KUKA KRL program: EPS_2_251825_SA13_A_20260116064054.src

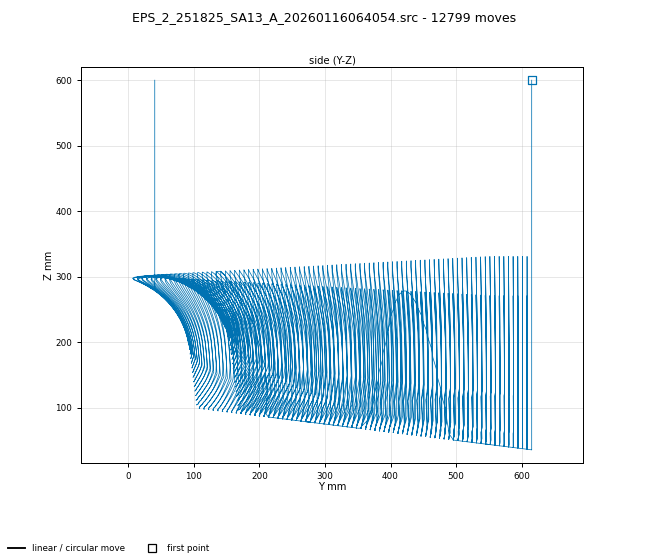
[picture p0: tool path of EPS_2_251825_SA13_A_20260116064054.src, 12799 of 12801 moves have a stored position in this frame; points joined in program order, loops and branches not executed]
&ACCESS RVP
&REL 4
&COMMENT QRS 19112012
&PARAM EDITMASK = *
DEF PART()
EXT BAS (BAS_COMMAND :IN,REAL :IN )
INT I
BAS (#INITMOV,0 )

;KUKA QRS Post kuka4.cps  Date:22-06-2017 !

File_ID=2975

QRS_PRE_INIT()

;Init var - Until changes are made in qrs_pre_init
Outlet_Square_prg=0
Inlet_1_Square_prg=0
Inlet_2_Square_prg=0
Inlet_3_Square_prg=0
Inlet_4_Square_prg=0
Inlet_5_Square_prg=0

Outlet_1={X 0.000, Y 551.740, Z 230.500, B 0.000, E1 0.000 }
Inlet_1={X 0.000, Y 556.010, Z 170.500, B 0.000, E1 170.000 }
Outlet_1_type=201
Inlet_1_type=201
;QRS#1=Sidecore dimensions
;QRS#2=200-8" PVC SDR 35
;QRS#3=200-8" PVC SDR 35
;QRS#4=
;QRS#5=
;QRS#6=
;QRS#7=
;QRS#8=
;QRS#9=12-08 PSX
;QRS#10=12-08 PSX
;QRS#11=
;QRS#12=
;QRS#13=
;QRS#14=
;QRS#15=
;QRS#16=1220x127x610 2'
;QRS#17=EPS Height
;QRS#18=331
;QRS#19=*
;QRS#20= UPDATED VERSION 22-06-2017
;QRS#21=*
Outlet_Square=0100
Inlet_1_Square=0100
Inlet_2_Square=0
Inlet_3_Square=0
Inlet_4_Square=0
Inlet_5_Square=0
Mill_Square=1
Outlet_Square_Prg=204
Inlet_1_Square_prg=204

QRS_INIT()

$ADVANCE=5

; T1
PTP {E1 173.62,E2 173.62}
PTP {X 0,Y 615.489,A -85,B 0,C 180,E1 173.62,E2 173.62,E3 0,E4 0,E5 0,E6 0}
QRS_SPEED_INIT()
LIN {X 0,Y 615.489,Z 600,A -85,B 0,C 180,E1 173.62,E2 173.62,E3 0,E4 0,E5 0,E6 0} C_VEL
LIN {X 0,Y 615.489,Z 45.866,A -85,B 0,C 180,E1 173.62,E2 173.62} C_VEL
LIN {X 0,Y 615.489,Z 37.686,A -85,B 0,C 180,E1 173.62,E2 173.62} C_VEL
LIN {X 0,Y 615.477,Z 35.686,A -85,B 0,C 180,E1 173.434,E2 173.434} C_VEL
LIN {X 0,Y 615.485,Z 35.695,A -85,B 0,C 180,E1 170.801,E2 170.801} C_VEL
LIN {X 0,Y 615.464,Z 35.693,A -85,B 0,C 180,E1 168.139,E2 168.139} C_VEL
LIN {X 0,Y 615.491,Z 35.685,A -85,B 0,C 180,E1 165.451,E2 165.451} C_VEL
LIN {X 0,Y 615.483,Z 35.698,A -85,B 0,C 180,E1 162.729,E2 162.729} C_VEL
LIN {X 0,Y 615.474,Z 35.687,A -85,B 0,C 180,E1 159.967,E2 159.967} C_VEL
LIN {X 0,Y 615.488,Z 35.701,A -85,B 0,C 180,E1 157.156,E2 157.156} C_VEL
LIN {X 0,Y 615.46,Z 35.69,A -85,B 0,C 180,E1 154.437,E2 154.437} C_VEL
LIN {X 0,Y 615.491,Z 35.695,A -85,B 0,C 180,E1 151.55,E2 151.55} C_VEL
LIN {X 0,Y 615.46,Z 35.694,A -85,B 0,C 180,E1 148.919,E2 148.919} C_VEL
LIN {X 0,Y 615.467,Z 35.688,A -85,B 0,C 180,E1 146.469,E2 146.469} C_VEL
LIN {X 0,Y 615.483,Z 35.701,A -85,B 0,C 180,E1 143.575,E2 143.575} C_VEL
LIN {X 0,Y 615.454,Z 35.692,A -85,B 0,C 180,E1 140.942,E2 140.942} C_VEL
LIN {X 0,Y 615.481,Z 35.687,A -85,B 0,C 180,E1 138.526,E2 138.526} C_VEL
LIN {X 0,Y 615.485,Z 35.699,A -85,B 0,C 180,E1 135.85,E2 135.85} C_VEL
LIN {X 0,Y 615.45,Z 35.692,A -85,B 0,C 180,E1 133.248,E2 133.248} C_VEL
LIN {X 0,Y 615.488,Z 35.69,A -85,B 0,C 180,E1 130.607,E2 130.607} C_VEL
LIN {X 0,Y 615.468,Z 35.698,A -85,B 0,C 180,E1 128.01,E2 128.01} C_VEL
LIN {X 0,Y 615.446,Z 35.694,A -85,B 0,C 180,E1 125.619,E2 125.619} C_VEL
LIN {X 0,Y 615.463,Z 35.69,A -85,B 0,C 180,E1 123.238,E2 123.238} C_VEL
LIN {X 0,Y 615.49,Z 35.692,A -85,B 0,C 180,E1 120.92,E2 120.92} C_VEL
LIN {X 0,Y 615.47,Z 35.699,A -85,B 0,C 180,E1 118.447,E2 118.447} C_VEL
LIN {X 0,Y 615.47,Z 35.794,A -85,B 0,C 180,E1 117.293,E2 117.293} C_VEL
LIN {X 0,Y 615.455,Z 50.485,A -85,B 0,C 180,E1 114.633,E2 114.633} C_VEL
LIN {X 0,Y 615.477,Z 60.616,A -85,B 0,C 180,E1 112.814,E2 112.814} C_VEL
LIN {X 0,Y 615.485,Z 166.964,A -85,B 0,C 180,E1 111.542,E2 111.542} C_VEL
LIN {X 0,Y 615.489,Z 179.954,A -85,B 0,C 180,E1 111.256,E2 111.256} C_VEL
LIN {X 0,Y 615.494,Z 193.256,A -85,B 0,C 180,E1 110.818,E2 110.818} C_VEL
LIN {X 0,Y 615.466,Z 204.889,A -85,B 0,C 180,E1 110.294,E2 110.294} C_VEL
LIN {X 0,Y 615.47,Z 215.474,A -85,B 0,C 180,E1 109.686,E2 109.686} C_VEL
LIN {X 0,Y 615.499,Z 226.345,A -85,B 0,C 180,E1 108.905,E2 108.905} C_VEL
LIN {X 0,Y 615.496,Z 235.253,A -85,B 0,C 180,E1 108.119,E2 108.119} C_VEL
LIN {X 0,Y 615.496,Z 244.551,A -85,B 0,C 180,E1 107.099,E2 107.099} C_VEL
LIN {X 0,Y 615.496,Z 251.406,A -85,B 0,C 180,E1 106.169,E2 106.169} C_VEL
LIN {X 0,Y 615.497,Z 257.042,A -85,B 0,C 180,E1 105.226,E2 105.226} C_VEL
LIN {X 0,Y 615.496,Z 261.719,A -85,B 0,C 180,E1 104.242,E2 104.242} C_VEL
LIN {X 0,Y 615.497,Z 265.484,A -85,B 0,C 180,E1 103.201,E2 103.201} C_VEL
LIN {X 0,Y 615.494,Z 267.337,A -85,B 0,C 180,E1 102.53,E2 102.53} C_VEL
LIN {X 0,Y 615.496,Z 268.704,A -85,B 0,C 180,E1 101.861,E2 101.861} C_VEL
LIN {X 0,Y 615.496,Z 270.232,A -85,B 0,C 180,E1 100.527,E2 100.527} C_VEL
LIN {X 0,Y 615.498,Z 270.372,A -85,B 0,C 180,E1 99.862,E2 99.862} C_VEL
LIN {X 0,Y 615.496,Z 269.451,A -85,B 0,C 180,E1 98.537,E2 98.537} C_VEL
LIN {X 0,Y 615.495,Z 268.407,A -85,B 0,C 180,E1 97.876,E2 97.876} C_VEL
LIN {X 0,Y 615.495,Z 265.082,A -85,B 0,C 180,E1 96.583,E2 96.583} C_VEL
LIN {X 0,Y 615.496,Z 261.297,A -85,B 0,C 180,E1 95.57,E2 95.57} C_VEL
LIN {X 0,Y 615.498,Z 256.495,A -85,B 0,C 180,E1 94.584,E2 94.584} C_VEL
LIN {X 0,Y 615.496,Z 250.457,A -85,B 0,C 180,E1 93.601,E2 93.601} C_VEL
LIN {X 0,Y 615.498,Z 242.969,A -85,B 0,C 180,E1 92.618,E2 92.618} C_VEL
LIN {X 0,Y 615.497,Z 235.341,A -85,B 0,C 180,E1 91.799,E2 91.799} C_VEL
LIN {X 0,Y 615.498,Z 225,A -85,B 0,C 180,E1 90.9,E2 90.9} C_VEL
LIN {X 0,Y 615.494,Z 214.531,A -85,B 0,C 180,E1 90.164,E2 90.164} C_VEL
LIN {X 0,Y 615.486,Z 204.413,A -85,B 0,C 180,E1 89.591,E2 89.591} C_VEL
LIN {X 0,Y 615.481,Z 192.391,A -85,B 0,C 180,E1 89.059,E2 89.059} C_VEL
LIN {X 0,Y 615.465,Z 179.856,A -85,B 0,C 180,E1 88.65,E2 88.65} C_VEL
LIN {X 0,Y 615.472,Z 166.761,A -85,B 0,C 180,E1 88.364,E2 88.364} C_VEL
LIN {X 0,Y 615.449,Z 60.618,A -85,B 0,C 180,E1 87.095,E2 87.095} C_VEL
LIN {X 0,Y 615.494,Z 45.776,A -85,B 0,C 180,E1 84.43,E2 84.43} C_VEL
LIN {X 0,Y 615.483,Z 35.688,A -85,B 0,C 180,E1 82.578,E2 82.578} C_VEL
LIN {X 0,Y 615.486,Z 35.684,A -85,B 0,C 180,E1 80.138,E2 80.138} C_VEL
LIN {X 0,Y 615.491,Z 35.698,A -85,B 0,C 180,E1 77.47,E2 77.47} C_VEL
LIN {X 0,Y 615.484,Z 35.686,A -85,B 0,C 180,E1 74.774,E2 74.774} C_VEL
LIN {X 0,Y 615.476,Z 35.691,A -85,B 0,C 180,E1 72.043,E2 72.043} C_VEL
LIN {X 0,Y 615.481,Z 35.692,A -85,B 0,C 180,E1 69.269,E2 69.269} C_VEL
LIN {X 0,Y 615.48,Z 35.687,A -85,B 0,C 180,E1 66.443,E2 66.443} C_VEL
LIN {X 0,Y 615.477,Z 35.691,A -85,B 0,C 180,E1 64.284,E2 64.284} C_VEL
LIN {X 0,Y 615.48,Z 35.693,A -85,B 0,C 180,E1 61.551,E2 61.551} C_VEL
LIN {X 0,Y 615.484,Z 35.684,A -85,B 0,C 180,E1 58.915,E2 58.915} C_VEL
LIN {X 0,Y 615.486,Z 35.698,A -85,B 0,C 180,E1 55.978,E2 55.978} C_VEL
LIN {X 0,Y 615.482,Z 35.685,A -85,B 0,C 180,E1 53.064,E2 53.064} C_VEL
LIN {X 0,Y 615.493,Z 35.698,A -85,B 0,C 180,E1 50.25,E2 50.25} C_VEL
LIN {X 0,Y 615.484,Z 35.685,A -85,B 0,C 180,E1 47.646,E2 47.646} C_VEL
LIN {X 0,Y 615.48,Z 35.692,A -85,B 0,C 180,E1 44.93,E2 44.93} C_VEL
LIN {X 0,Y 615.477,Z 35.69,A -85,B 0,C 180,E1 42.078,E2 42.078} C_VEL
LIN {X 0,Y 615.494,Z 35.682,A -85,B 0,C 180,E1 39.75,E2 39.75} C_VEL
LIN {X 0,Y 615.484,Z 35.699,A -85,B 0,C 180,E1 36.935,E2 36.935} C_VEL
LIN {X 0,Y 615.485,Z 35.696,A -85,B 0,C 180,E1 34.7,E2 34.7} C_VEL
LIN {X 0,Y 615.473,Z 35.689,A -85,B 0,C 180,E1 32.328,E2 32.328} C_VEL
LIN {X 0,Y 615.487,Z 35.685,A -85,B 0,C 180,E1 29.794,E2 29.794} C_VEL
LIN {X 0,Y 615.49,Z 35.698,A -85,B 0,C 180,E1 27.044,E2 27.044} C_VEL
LIN {X 0,Y 615.487,Z 35.683,A -85,B 0,C 180,E1 24.272,E2 24.272} C_VEL
LIN {X 0,Y 615.494,Z 35.699,A -85,B 0,C 180,E1 21.432,E2 21.432} C_VEL
LIN {X 0,Y 615.483,Z 35.684,A -85,B 0,C 180,E1 18.602,E2 18.602} C_VEL
LIN {X 0,Y 615.484,Z 35.693,A -85,B 0,C 180,E1 15.905,E2 15.905} C_VEL
LIN {X 0,Y 615.474,Z 35.692,A -85,B 0,C 180,E1 13.201,E2 13.201} C_VEL
LIN {X 0,Y 615.487,Z 35.684,A -85,B 0,C 180,E1 10.527,E2 10.527} C_VEL
LIN {X 0,Y 615.487,Z 35.703,A -85,B 0,C 180,E1 7.876,E2 7.876} C_VEL
LIN {X 0,Y 615.474,Z 35.688,A -85,B 0,C 180,E1 5.241,E2 5.241} C_VEL
LIN {X 0,Y 615.486,Z 35.687,A -85,B 0,C 180,E1 2.618,E2 2.618} C_VEL
LIN {X 0,Y 615.486,Z 35.698,A -85,B 0,C 180,E1 0,E2 0} C_VEL
LIN {X 0,Y 615.478,Z 35.686,A -85,B 0,C 180,E1 -2.618,E2 -2.618} C_VEL
LIN {X 0,Y 615.485,Z 35.69,A -85,B 0,C 180,E1 -5.241,E2 -5.241} C_VEL
LIN {X 0,Y 615.477,Z 35.695,A -85,B 0,C 180,E1 -7.876,E2 -7.876} C_VEL
LIN {X 0,Y 615.484,Z 35.684,A -85,B 0,C 180,E1 -10.527,E2 -10.527} C_VEL
LIN {X 0,Y 615.49,Z 35.696,A -85,B 0,C 180,E1 -13.201,E2 -13.201} C_VEL
LIN {X 0,Y 615.469,Z 35.69,A -85,B 0,C 180,E1 -15.906,E2 -15.906} C_VEL
LIN {X 0,Y 615.487,Z 35.688,A -85,B 0,C 180,E1 -18.646,E2 -18.646} C_VEL
LIN {X 0,Y 615.474,Z 35.695,A -85,B 0,C 180,E1 -21.433,E2 -21.433} C_VEL
LIN {X 0,Y 615.49,Z 35.684,A -85,B 0,C 180,E1 -24.272,E2 -24.272} C_VEL
LIN {X 0,Y 615.475,Z 35.696,A -85,B 0,C 180,E1 -27.178,E2 -27.178} C_VEL
LIN {X 0,Y 615.481,Z 35.685,A -85,B 0,C 180,E1 -29.793,E2 -29.793} C_VEL
LIN {X 0,Y 615.489,Z 35.695,A -85,B 0,C 180,E1 -32.458,E2 -32.458} C_VEL
LIN {X 0,Y 615.478,Z 35.697,A -85,B 0,C 180,E1 -34.816,E2 -34.816} C_VEL
LIN {X 0,Y 615.467,Z 35.689,A -85,B 0,C 180,E1 -37.244,E2 -37.244} C_VEL
LIN {X 0,Y 615.487,Z 35.693,A -85,B 0,C 180,E1 -40.088,E2 -40.088} C_VEL
LIN {X 0,Y 615.497,Z 35.7,A -85,B 0,C 180,E1 -42.352,E2 -42.352} C_VEL
LIN {X 0,Y 615.469,Z 35.688,A -85,B 0,C 180,E1 -45.071,E2 -45.071} C_VEL
LIN {X 0,Y 615.491,Z 35.695,A -85,B 0,C 180,E1 -47.92,E2 -47.92} C_VEL
LIN {X 0,Y 615.479,Z 35.697,A -85,B 0,C 180,E1 -50.249,E2 -50.249} C_VEL
LIN {X 0,Y 615.478,Z 35.686,A -85,B 0,C 180,E1 -53.065,E2 -53.065} C_VEL
LIN {X 0,Y 615.486,Z 35.698,A -85,B 0,C 180,E1 -55.978,E2 -55.978} C_VEL
LIN {X 0,Y 615.46,Z 35.693,A -85,B 0,C 180,E1 -58.313,E2 -58.313} C_VEL
LIN {X 0,Y 615.469,Z 35.688,A -85,B 0,C 180,E1 -60.592,E2 -60.592} C_VEL
LIN {X 0,Y 615.492,Z 35.702,A -85,B 0,C 180,E1 -63.556,E2 -63.556} C_VEL
LIN {X 0,Y 615.463,Z 35.693,A -85,B 0,C 180,E1 -65.997,E2 -65.997} C_VEL
LIN {X 0,Y 615.484,Z 35.871,A -85,B 0,C 180,E1 -66.711,E2 -66.711} C_VEL
LIN {X 0,Y 615.45,Z 57.104,A -85,B 0,C 180,E1 -69.453,E2 -69.453} C_VEL
LIN {X 0,Y 615.489,Z 77.472,A -85,B 0,C 180,E1 -72.043,E2 -72.043} C_VEL
LIN {X 0,Y 615.495,Z 99.259,A -85,B 0,C 180,E1 -74.774,E2 -74.774} C_VEL
LIN {X 0,Y 615.459,Z 118.134,A -85,B 0,C 180,E1 -77.113,E2 -77.113} C_VEL
LIN {X 0,Y 615.491,Z 226.821,A -85,B 0,C 180,E1 -78.411,E2 -78.411} C_VEL
LIN {X 0,Y 615.484,Z 239.339,A -85,B 0,C 180,E1 -78.682,E2 -78.682} C_VEL
LIN {X 0,Y 615.49,Z 252.594,A -85,B 0,C 180,E1 -79.112,E2 -79.112} C_VEL
LIN {X 0,Y 615.473,Z 264.477,A -85,B 0,C 180,E1 -79.639,E2 -79.639} C_VEL
LIN {X 0,Y 615.49,Z 275.992,A -85,B 0,C 180,E1 -80.304,E2 -80.304} C_VEL
LIN {X 0,Y 615.499,Z 286.339,A -85,B 0,C 180,E1 -81.05,E2 -81.05} C_VEL
LIN {X 0,Y 615.497,Z 294.81,A -85,B 0,C 180,E1 -81.794,E2 -81.794} C_VEL
LIN {X 0,Y 615.498,Z 302.605,A -85,B 0,C 180,E1 -82.619,E2 -82.619} C_VEL
LIN {X 0,Y 615.496,Z 310.202,A -85,B 0,C 180,E1 -83.608,E2 -83.608} C_VEL
LIN {X 0,Y 615.498,Z 317.204,A -85,B 0,C 180,E1 -84.759,E2 -84.759} C_VEL
LIN {X 0,Y 615.493,Z 321.851,A -85,B 0,C 180,E1 -85.743,E2 -85.743} C_VEL
LIN {X 0,Y 615.494,Z 325.398,A -85,B 0,C 180,E1 -86.727,E2 -86.727} C_VEL
LIN {X 0,Y 615.497,Z 327.233,A -85,B 0,C 180,E1 -87.382,E2 -87.382} C_VEL
LIN {X 0,Y 615.5,Z 328.607,A -85,B 0,C 180,E1 -88.037,E2 -88.037} C_VEL
LIN {X 0,Y 615.496,Z 330.173,A -85,B 0,C 180,E1 -89.346,E2 -89.346} C_VEL
LIN {X 0,Y 615.494,Z 330.389,A -85,B 0,C 180,E1 -90,E2 -90} C_VEL
LIN {X 0,Y 615.495,Z 329.58,A -85,B 0,C 180,E1 -91.309,E2 -91.309} C_VEL
LIN {X 0,Y 615.5,Z 328.608,A -85,B 0,C 180,E1 -91.963,E2 -91.963} C_VEL
LIN {X 0,Y 615.497,Z 327.233,A -85,B 0,C 180,E1 -92.618,E2 -92.618} C_VEL
LIN {X 0,Y 615.496,Z 324.349,A -85,B 0,C 180,E1 -93.601,E2 -93.601} C_VEL
LIN {X 0,Y 615.498,Z 320.441,A -85,B 0,C 180,E1 -94.584,E2 -94.584} C_VEL
LIN {X 0,Y 615.499,Z 315.405,A -85,B 0,C 180,E1 -95.57,E2 -95.57} C_VEL
LIN {X 0,Y 615.497,Z 308.87,A -85,B 0,C 180,E1 -96.583,E2 -96.583} C_VEL
LIN {X 0,Y 615.497,Z 301.133,A -85,B 0,C 180,E1 -97.545,E2 -97.545} C_VEL
LIN {X 0,Y 615.498,Z 293.045,A -85,B 0,C 180,E1 -98.371,E2 -98.371} C_VEL
LIN {X 0,Y 615.499,Z 283.167,A -85,B 0,C 180,E1 -99.199,E2 -99.199} C_VEL
LIN {X 0,Y 615.48,Z 271.982,A -85,B 0,C 180,E1 -99.945,E2 -99.945} C_VEL
LIN {X 0,Y 615.48,Z 261.023,A -85,B 0,C 180,E1 -100.527,E2 -100.527} C_VEL
LIN {X 0,Y 615.484,Z 248.476,A -85,B 0,C 180,E1 -101.041,E2 -101.041} C_VEL
LIN {X 0,Y 615.482,Z 236.064,A -85,B 0,C 180,E1 -101.402,E2 -101.402} C_VEL
LIN {X 0,Y 615.494,Z 222.461,A -85,B 0,C 180,E1 -101.652,E2 -101.652} C_VEL
LIN {X 0,Y 615.459,Z 118.134,A -85,B 0,C 180,E1 -102.887,E2 -102.887} C_VEL
LIN {X 0,Y 615.479,Z 95.176,A -85,B 0,C 180,E1 -105.735,E2 -105.735} C_VEL
LIN {X 0,Y 615.474,Z 73.67,A -85,B 0,C 180,E1 -108.438,E2 -108.438} C_VEL
LIN {X 0,Y 615.491,Z 51.566,A -85,B 0,C 180,E1 -111.256,E2 -111.256} C_VEL
LIN {X 0,Y 615.485,Z 35.685,A -85,B 0,C 180,E1 -113.334,E2 -113.334} C_VEL
LIN {X 0,Y 615.464,Z 35.69,A -85,B 0,C 180,E1 -115.717,E2 -115.717} C_VEL
LIN {X 0,Y 615.494,Z 35.697,A -85,B 0,C 180,E1 -118.451,E2 -118.451} C_VEL
LIN {X 0,Y 615.481,Z 35.685,A -85,B 0,C 180,E1 -121.085,E2 -121.085} C_VEL
LIN {X 0,Y 615.466,Z 35.691,A -85,B 0,C 180,E1 -123.531,E2 -123.531} C_VEL
LIN {X 0,Y 615.482,Z 35.697,A -85,B 0,C 180,E1 -125.833,E2 -125.833} C_VEL
LIN {X 0,Y 615.487,Z 35.699,A -85,B 0,C 180,E1 -128.069,E2 -128.069} C_VEL
LIN {X 0,Y 615.486,Z 35.685,A -85,B 0,C 180,E1 -130.607,E2 -130.607} C_VEL
LIN {X 0,Y 615.471,Z 35.692,A -85,B 0,C 180,E1 -133.246,E2 -133.246} C_VEL
LIN {X 0,Y 615.485,Z 35.692,A -85,B 0,C 180,E1 -136.003,E2 -136.003} C_VEL
LIN {X 0,Y 615.486,Z 35.684,A -85,B 0,C 180,E1 -138.526,E2 -138.526} C_VEL
LIN {X 0,Y 615.478,Z 35.695,A -85,B 0,C 180,E1 -141.095,E2 -141.095} C_VEL
LIN {X 0,Y 615.486,Z 35.695,A -85,B 0,C 180,E1 -143.575,E2 -143.575} C_VEL
LIN {X 0,Y 615.486,Z 35.685,A -85,B 0,C 180,E1 -145.978,E2 -145.978} C_VEL
LIN {X 0,Y 615.482,Z 35.698,A -85,B 0,C 180,E1 -148.916,E2 -148.916} C_VEL
LIN {X 0,Y 615.481,Z 35.689,A -85,B 0,C 180,E1 -151.552,E2 -151.552} C_VEL
LIN {X 0,Y 615.478,Z 35.689,A -85,B 0,C 180,E1 -154.284,E2 -154.284} C_VEL
LIN {X 0,Y 615.48,Z 35.693,A -85,B 0,C 180,E1 -156.443,E2 -156.443} C_VEL
LIN {X 0,Y 615.478,Z 35.689,A -85,B 0,C 180,E1 -159.269,E2 -159.269} C_VEL
LIN {X 0,Y 615.48,Z 35.69,A -85,B 0,C 180,E1 -162.043,E2 -162.043} C_VEL
LIN {X 0,Y 615.479,Z 35.694,A -85,B 0,C 180,E1 -164.774,E2 -164.774} C_VEL
LIN {X 0,Y 615.491,Z 35.683,A -85,B 0,C 180,E1 -167.47,E2 -167.47} C_VEL
LIN {X 0,Y 615.494,Z 35.698,A -85,B 0,C 180,E1 -170.138,E2 -170.138} C_VEL
LIN {X 0,Y 615.474,Z 35.689,A -85,B 0,C 180,E1 -172.784,E2 -172.784} C_VEL
LIN {X 0,Y 615.487,Z 35.687,A -85,B 0,C 180,E1 -175.415,E2 -175.415} C_VEL
LIN {X 0,Y 615.488,Z 35.698,A -85,B 0,C 180,E1 -178.037,E2 -178.037} C_VEL
LIN {X 0,Y 615.476,Z 35.686,A -85,B 0,C 180,E1 -180.654,E2 -180.654} C_VEL
LIN {X 0,Y 615.484,Z 35.691,A -85,B 0,C 180,E1 -183.273,E2 -183.273} C_VEL
LIN {X 0,Y 615.473,Z 35.696,A -85,B 0,C 180,E1 -185.899,E2 -185.899} C_VEL
LIN {X 0,Y 615.477,Z 35.686,A -85,B 0,C 180,E1 -186.566,E2 -186.566} C_VEL
LIN {X 0,Y 614.809,Z 35.84,A -85,B 0,C 180,E1 -187.112,E2 -187.112} C_VEL
LIN {X 0,Y 611.981,Z 36.251,A -85,B 0,C 180,E1 -187.998,E2 -187.998} C_VEL
LIN {X 0,Y 609.588,Z 36.566,A -85,B 0,C 180,E1 -188.711,E2 -188.711} C_VEL
LIN {X 0,Y 608.547,Z 36.685,A -85,B 0,C 180,E1 -189.26,E2 -189.26} C_VEL
LIN {X 0,Y 608.455,Z 36.693,A -85,B 0,C 180,E1 -189.447,E2 -189.447} C_VEL
LIN {X 0,Y 608.448,Z 36.69,A -85,B 0,C 180,E1 -192,E2 -192} C_VEL
LIN {X 0,Y 608.48,Z 36.687,A -85,B 0,C 180,E1 -194.72,E2 -194.72} C_VEL
LIN {X 0,Y 608.446,Z 36.693,A -85,B 0,C 180,E1 -197.477,E2 -197.477} C_VEL
LIN {X 0,Y 608.441,Z 36.691,A -85,B 0,C 180,E1 -199.571,E2 -199.571} C_VEL
LIN {X 0,Y 608.482,Z 36.687,A -85,B 0,C 180,E1 -202.405,E2 -202.405} C_VEL
LIN {X 0,Y 608.454,Z 36.694,A -85,B 0,C 180,E1 -204.571,E2 -204.571} C_VEL
LIN {X 0,Y 608.438,Z 36.69,A -85,B 0,C 180,E1 -207.519,E2 -207.519} C_VEL
LIN {X 0,Y 608.465,Z 36.688,A -85,B 0,C 180,E1 -209.97,E2 -209.97} C_VEL
LIN {X 0,Y 608.447,Z 36.692,A -85,B 0,C 180,E1 -212.88,E2 -212.88} C_VEL
LIN {X 0,Y 608.43,Z 36.691,A -85,B 0,C 180,E1 -215.279,E2 -215.279} C_VEL
LIN {X 0,Y 608.469,Z 36.696,A -85,B 0,C 180,E1 -218.24,E2 -218.24} C_VEL
LIN {X 0,Y 608.448,Z 36.689,A -85,B 0,C 180,E1 -221.34,E2 -221.34} C_VEL
LIN {X 0,Y 608.452,Z 36.694,A -85,B 0,C 180,E1 -224.263,E2 -224.263} C_VEL
LIN {X 0,Y 608.428,Z 36.691,A -85,B 0,C 180,E1 -227.038,E2 -227.038} C_VEL
LIN {X 0,Y 608.455,Z 36.696,A -85,B 0,C 180,E1 -229.697,E2 -229.697} C_VEL
LIN {X 0,Y 608.45,Z 36.69,A -85,B 0,C 180,E1 -232.252,E2 -232.252} C_VEL
LIN {X 0,Y 608.456,Z 36.69,A -85,B 0,C 180,E1 -235.094,E2 -235.094} C_VEL
LIN {X 0,Y 608.448,Z 36.692,A -85,B 0,C 180,E1 -237.904,E2 -237.904} C_VEL
LIN {X 0,Y 608.43,Z 36.691,A -85,B 0,C 180,E1 -240.218,E2 -240.218} C_VEL
LIN {X 0,Y 608.457,Z 36.841,A -85,B 0,C 180,E1 -242.674,E2 -242.674} C_VEL
LIN {X 0,Y 608.437,Z 51.932,A -85,B 0,C 180,E1 -245.428,E2 -245.428} C_VEL
LIN {X 0,Y 608.44,Z 60.876,A -85,B 0,C 180,E1 -247.044,E2 -247.044} C_VEL
LIN {X 0,Y 608.538,Z 167.581,A -85,B 0,C 180,E1 -248.333,E2 -248.333} C_VEL
LIN {X 0,Y 608.54,Z 181.203,A -85,B 0,C 180,E1 -248.644,E2 -248.644} C_VEL
LIN {X 0,Y 608.54,Z 193.758,A -85,B 0,C 180,E1 -249.07,E2 -249.07} C_VEL
LIN {X 0,Y 608.473,Z 205.208,A -85,B 0,C 180,E1 -249.594,E2 -249.594} C_VEL
LIN {X 0,Y 608.477,Z 216.479,A -85,B 0,C 180,E1 -250.254,E2 -250.254} C_VEL
LIN {X 0,Y 608.473,Z 227.262,A -85,B 0,C 180,E1 -251.043,E2 -251.043} C_VEL
LIN {X 0,Y 608.465,Z 235.987,A -85,B 0,C 180,E1 -251.829,E2 -251.829} C_VEL
LIN {X 0,Y 608.457,Z 245.346,A -85,B 0,C 180,E1 -252.87,E2 -252.87} C_VEL
LIN {X 0,Y 608.458,Z 252.813,A -85,B 0,C 180,E1 -253.906,E2 -253.906} C_VEL
LIN {X 0,Y 608.439,Z 258.69,A -85,B 0,C 180,E1 -254.936,E2 -254.936} C_VEL
LIN {X 0,Y 608.442,Z 263.388,A -85,B 0,C 180,E1 -255.994,E2 -255.994} C_VEL
LIN {X 0,Y 608.446,Z 265.665,A -85,B 0,C 180,E1 -256.643,E2 -256.643} C_VEL
LIN {X 0,Y 608.419,Z 267.611,A -85,B 0,C 180,E1 -257.322,E2 -257.322} C_VEL
LIN {X 0,Y 608.44,Z 269.102,A -85,B 0,C 180,E1 -258,E2 -258} C_VEL
LIN {X 0,Y 608.437,Z 270.76,A -85,B 0,C 180,E1 -259.35,E2 -259.35} C_VEL
LIN {X 0,Y 608.433,Z 270.999,A -85,B 0,C 180,E1 -260.022,E2 -260.022} C_VEL
LIN {X 0,Y 608.421,Z 270.793,A -85,B 0,C 180,E1 -260.693,E2 -260.693} C_VEL
LIN {X 0,Y 608.42,Z 269.199,A -85,B 0,C 180,E1 -262.032,E2 -262.032} C_VEL
LIN {X 0,Y 608.424,Z 267.792,A -85,B 0,C 180,E1 -262.7,E2 -262.7} C_VEL
LIN {X 0,Y 608.452,Z 265.088,A -85,B 0,C 180,E1 -263.628,E2 -263.628} C_VEL
LIN {X 0,Y 608.44,Z 260.884,A -85,B 0,C 180,E1 -264.698,E2 -264.698} C_VEL
LIN {X 0,Y 608.437,Z 254.79,A -85,B 0,C 180,E1 -265.86,E2 -265.86} C_VEL
LIN {X 0,Y 608.458,Z 248.157,A -85,B 0,C 180,E1 -266.855,E2 -266.855} C_VEL
LIN {X 0,Y 608.454,Z 239.958,A -85,B 0,C 180,E1 -267.849,E2 -267.849} C_VEL
LIN {X 0,Y 608.482,Z 231.585,A -85,B 0,C 180,E1 -268.676,E2 -268.676} C_VEL
LIN {X 0,Y 608.476,Z 221.295,A -85,B 0,C 180,E1 -269.504,E2 -269.504} C_VEL
LIN {X 0,Y 608.5,Z 209.767,A -85,B 0,C 180,E1 -270.248,E2 -270.248} C_VEL
LIN {X 0,Y 608.534,Z 198.292,A -85,B 0,C 180,E1 -270.827,E2 -270.827} C_VEL
LIN {X 0,Y 608.521,Z 186.509,A -85,B 0,C 180,E1 -271.282,E2 -271.282} C_VEL
LIN {X 0,Y 608.511,Z 173.805,A -85,B 0,C 180,E1 -271.634,E2 -271.634} C_VEL
LIN {X 0,Y 608.533,Z 160.393,A -85,B 0,C 180,E1 -271.861,E2 -271.861} C_VEL
LIN {X 0,Y 608.409,Z 60.903,A -85,B 0,C 180,E1 -273.042,E2 -273.042} C_VEL
LIN {X 0,Y 608.487,Z 44.75,A -85,B 0,C 180,E1 -275.967,E2 -275.967} C_VEL
LIN {X 0,Y 608.46,Z 36.689,A -85,B 0,C 180,E1 -277.466,E2 -277.466} C_VEL
LIN {X 0,Y 608.455,Z 36.688,A -85,B 0,C 180,E1 -279.977,E2 -279.977} C_VEL
LIN {X 0,Y 608.477,Z 36.695,A -85,B 0,C 180,E1 -282.677,E2 -282.677} C_VEL
LIN {X 0,Y 608.468,Z 36.686,A -85,B 0,C 180,E1 -285.406,E2 -285.406} C_VEL
LIN {X 0,Y 608.443,Z 36.695,A -85,B 0,C 180,E1 -288.172,E2 -288.172} C_VEL
LIN {X 0,Y 608.455,Z 36.689,A -85,B 0,C 180,E1 -290.982,E2 -290.982} C_VEL
LIN {X 0,Y 608.446,Z 36.689,A -85,B 0,C 180,E1 -293.124,E2 -293.124} C_VEL
LIN {X 0,Y 608.465,Z 36.689,A -85,B 0,C 180,E1 -295.719,E2 -295.719} C_VEL
LIN {X 0,Y 608.448,Z 36.695,A -85,B 0,C 180,E1 -298.267,E2 -298.267} C_VEL
LIN {X 0,Y 608.474,Z 36.687,A -85,B 0,C 180,E1 -300.545,E2 -300.545} C_VEL
LIN {X 0,Y 608.452,Z 36.688,A -85,B 0,C 180,E1 -302.88,E2 -302.88} C_VEL
LIN {X 0,Y 608.445,Z 36.691,A -85,B 0,C 180,E1 -305.278,E2 -305.278} C_VEL
LIN {X 0,Y 608.465,Z 36.697,A -85,B 0,C 180,E1 -307.747,E2 -307.747} C_VEL
LIN {X 0,Y 608.447,Z 36.689,A -85,B 0,C 180,E1 -310.328,E2 -310.328} C_VEL
LIN {X 0,Y 608.471,Z 36.692,A -85,B 0,C 180,E1 -313.309,E2 -313.309} C_VEL
LIN {X 0,Y 608.464,Z 36.687,A -85,B 0,C 180,E1 -316.13,E2 -316.13} C_VEL
LIN {X 0,Y 608.451,Z 36.69,A -85,B 0,C 180,E1 -318.823,E2 -318.823} C_VEL
LIN {X 0,Y 608.463,Z 36.689,A -85,B 0,C 180,E1 -321.761,E2 -321.761} C_VEL
LIN {X 0,Y 608.45,Z 36.688,A -85,B 0,C 180,E1 -323.955,E2 -323.955} C_VEL
LIN {X 0,Y 608.45,Z 36.689,A -85,B 0,C 180,E1 -326.328,E2 -326.328} C_VEL
LIN {X 0,Y 608.449,Z 36.694,A -85,B 0,C 180,E1 -328.733,E2 -328.733} C_VEL
LIN {X 0,Y 608.464,Z 36.689,A -85,B 0,C 180,E1 -331.383,E2 -331.383} C_VEL
LIN {X 0,Y 608.44,Z 36.69,A -85,B 0,C 180,E1 -333.964,E2 -333.964} C_VEL
LIN {X 0,Y 608.468,Z 36.688,A -85,B 0,C 180,E1 -336.155,E2 -336.155} C_VEL
LIN {X 0,Y 608.455,Z 36.691,A -85,B 0,C 180,E1 -339.018,E2 -339.018} C_VEL
LIN {X 0,Y 608.446,Z 36.69,A -85,B 0,C 180,E1 -341.828,E2 -341.828} C_VEL
LIN {X 0,Y 608.464,Z 36.693,A -85,B 0,C 180,E1 -344.594,E2 -344.594} C_VEL
LIN {X 0,Y 608.476,Z 36.685,A -85,B 0,C 180,E1 -347.323,E2 -347.323} C_VEL
LIN {X 0,Y 608.464,Z 36.693,A -85,B 0,C 180,E1 -350.023,E2 -350.023} C_VEL
LIN {X 0,Y 608.443,Z 36.691,A -85,B 0,C 180,E1 -352.7,E2 -352.7} C_VEL
LIN {X 0,Y 608.454,Z 36.689,A -85,B 0,C 180,E1 -355.362,E2 -355.362} C_VEL
LIN {X 0,Y 608.459,Z 36.696,A -85,B 0,C 180,E1 -358.014,E2 -358.014} C_VEL
LIN {X 0,Y 608.473,Z 36.686,A -85,B 0,C 180,E1 -360.662,E2 -360.662} C_VEL
LIN {X 0,Y 608.477,Z 36.688,A -85,B 0,C 180,E1 -363.311,E2 -363.311} C_VEL
LIN {X 0,Y 608.454,Z 36.692,A -85,B 0,C 180,E1 -365.967,E2 -365.967} C_VEL
LIN {X 0,Y 608.456,Z 36.687,A -85,B 0,C 180,E1 -368.636,E2 -368.636} C_VEL
LIN {X 0,Y 608.461,Z 36.695,A -85,B 0,C 180,E1 -371.324,E2 -371.324} C_VEL
LIN {X 0,Y 608.452,Z 36.689,A -85,B 0,C 180,E1 -374.038,E2 -374.038} C_VEL
LIN {X 0,Y 608.48,Z 36.687,A -85,B 0,C 180,E1 -376.783,E2 -376.783} C_VEL
LIN {X 0,Y 608.448,Z 36.692,A -85,B 0,C 180,E1 -379.571,E2 -379.571} C_VEL
LIN {X 0,Y 608.465,Z 36.688,A -85,B 0,C 180,E1 -382.476,E2 -382.476} C_VEL
LIN {X 0,Y 608.458,Z 36.691,A -85,B 0,C 180,E1 -384.571,E2 -384.571} C_VEL
LIN {X 0,Y 608.445,Z 36.69,A -85,B 0,C 180,E1 -387.518,E2 -387.518} C_VEL
LIN {X 0,Y 608.467,Z 36.686,A -85,B 0,C 180,E1 -389.97,E2 -389.97} C_VEL
LIN {X 0,Y 608.45,Z 36.695,A -85,B 0,C 180,E1 -392.88,E2 -392.88} C_VEL
LIN {X 0,Y 608.437,Z 36.691,A -85,B 0,C 180,E1 -395.278,E2 -395.278} C_VEL
LIN {X 0,Y 608.467,Z 36.692,A -85,B 0,C 180,E1 -398.24,E2 -398.24} C_VEL
LIN {X 0,Y 608.453,Z 36.688,A -85,B 0,C 180,E1 -401.341,E2 -401.341} C_VEL
LIN {X 0,Y 608.46,Z 36.697,A -85,B 0,C 180,E1 -404.264,E2 -404.264} C_VEL
LIN {X 0,Y 608.437,Z 36.69,A -85,B 0,C 180,E1 -407.038,E2 -407.038} C_VEL
LIN {X 0,Y 608.457,Z 36.692,A -85,B 0,C 180,E1 -409.697,E2 -409.697} C_VEL
LIN {X 0,Y 608.463,Z 36.692,A -85,B 0,C 180,E1 -412.253,E2 -412.253} C_VEL
LIN {X 0,Y 608.458,Z 36.688,A -85,B 0,C 180,E1 -415.094,E2 -415.094} C_VEL
LIN {X 0,Y 608.464,Z 36.694,A -85,B 0,C 180,E1 -417.905,E2 -417.905} C_VEL
LIN {X 0,Y 608.45,Z 36.69,A -85,B 0,C 180,E1 -420.219,E2 -420.219} C_VEL
LIN {X 0,Y 608.482,Z 36.685,A -85,B 0,C 180,E1 -422.793,E2 -422.793} C_VEL
LIN {X 0,Y 608.464,Z 36.692,A -85,B 0,C 180,E1 -425.851,E2 -425.851} C_VEL
LIN {X 0,Y 608.51,Z 36.894,A -85,B 0,C 180,E1 -426.563,E2 -426.563} C_VEL
LIN {X 0,Y 608.569,Z 54.295,A -85,B 0,C 180,E1 -428.845,E2 -428.845} C_VEL
LIN {X 0,Y 608.537,Z 74.958,A -85,B 0,C 180,E1 -431.507,E2 -431.507} C_VEL
LIN {X 0,Y 608.489,Z 96.602,A -85,B 0,C 180,E1 -434.251,E2 -434.251} C_VEL
LIN {X 0,Y 608.456,Z 118.353,A -85,B 0,C 180,E1 -436.972,E2 -436.972} C_VEL
LIN {X 0,Y 608.547,Z 226.938,A -85,B 0,C 180,E1 -438.276,E2 -438.276} C_VEL
LIN {X 0,Y 608.519,Z 240.211,A -85,B 0,C 180,E1 -438.571,E2 -438.571} C_VEL
LIN {X 0,Y 608.516,Z 252.615,A -85,B 0,C 180,E1 -438.982,E2 -438.982} C_VEL
LIN {X 0,Y 608.497,Z 264.632,A -85,B 0,C 180,E1 -439.519,E2 -439.519} C_VEL
LIN {X 0,Y 608.477,Z 276.195,A -85,B 0,C 180,E1 -440.191,E2 -440.191} C_VEL
LIN {X 0,Y 608.485,Z 286.592,A -85,B 0,C 180,E1 -440.946,E2 -440.946} C_VEL
LIN {X 0,Y 608.475,Z 295.11,A -85,B 0,C 180,E1 -441.699,E2 -441.699} C_VEL
LIN {X 0,Y 608.471,Z 302.959,A -85,B 0,C 180,E1 -442.534,E2 -442.534} C_VEL
LIN {X 0,Y 608.461,Z 310.286,A -85,B 0,C 180,E1 -443.484,E2 -443.484} C_VEL
LIN {X 0,Y 608.451,Z 315.865,A -85,B 0,C 180,E1 -444.365,E2 -444.365} C_VEL
LIN {X 0,Y 608.432,Z 320.95,A -85,B 0,C 180,E1 -445.362,E2 -445.362} C_VEL
LIN {X 0,Y 608.449,Z 324.896,A -85,B 0,C 180,E1 -446.358,E2 -446.358} C_VEL
LIN {X 0,Y 608.425,Z 327.809,A -85,B 0,C 180,E1 -447.352,E2 -447.352} C_VEL
LIN {X 0,Y 608.444,Z 329.201,A -85,B 0,C 180,E1 -448.014,E2 -448.014} C_VEL
LIN {X 0,Y 608.438,Z 330.783,A -85,B 0,C 180,E1 -449.338,E2 -449.338} C_VEL
LIN {X 0,Y 608.434,Z 331,A -85,B 0,C 180,E1 -450,E2 -450} C_VEL
LIN {X 0,Y 608.448,Z 330.184,A -85,B 0,C 180,E1 -451.324,E2 -451.324} C_VEL
LIN {X 0,Y 608.444,Z 329.201,A -85,B 0,C 180,E1 -451.986,E2 -451.986} C_VEL
LIN {X 0,Y 608.425,Z 327.809,A -85,B 0,C 180,E1 -452.648,E2 -452.648} C_VEL
LIN {X 0,Y 608.449,Z 324.896,A -85,B 0,C 180,E1 -453.642,E2 -453.642} C_VEL
LIN {X 0,Y 608.432,Z 320.95,A -85,B 0,C 180,E1 -454.638,E2 -454.638} C_VEL
LIN {X 0,Y 608.438,Z 314.877,A -85,B 0,C 180,E1 -455.801,E2 -455.801} C_VEL
LIN {X 0,Y 608.462,Z 308.235,A -85,B 0,C 180,E1 -456.799,E2 -456.799} C_VEL
LIN {X 0,Y 608.456,Z 299.989,A -85,B 0,C 180,E1 -457.8,E2 -457.8} C_VEL
LIN {X 0,Y 608.472,Z 291.536,A -85,B 0,C 180,E1 -458.636,E2 -458.636} C_VEL
LIN {X 0,Y 608.48,Z 281.091,A -85,B 0,C 180,E1 -459.473,E2 -459.473} C_VEL
LIN {X 0,Y 608.484,Z 270.756,A -85,B 0,C 180,E1 -460.145,E2 -460.145} C_VEL
LIN {X 0,Y 608.519,Z 259.261,A -85,B 0,C 180,E1 -460.74,E2 -460.74} C_VEL
LIN {X 0,Y 608.531,Z 246.887,A -85,B 0,C 180,E1 -461.225,E2 -461.225} C_VEL
LIN {X 0,Y 608.546,Z 233.436,A -85,B 0,C 180,E1 -461.597,E2 -461.597} C_VEL
LIN {X 0,Y 608.552,Z 221.081,A -85,B 0,C 180,E1 -461.808,E2 -461.808} C_VEL
LIN {X 0,Y 608.445,Z 118.269,A -85,B 0,C 180,E1 -463.038,E2 -463.038} C_VEL
LIN {X 0,Y 608.495,Z 95.239,A -85,B 0,C 180,E1 -465.921,E2 -465.921} C_VEL
LIN {X 0,Y 608.537,Z 74.958,A -85,B 0,C 180,E1 -468.493,E2 -468.493} C_VEL
LIN {X 0,Y 608.569,Z 54.296,A -85,B 0,C 180,E1 -471.155,E2 -471.155} C_VEL
LIN {X 0,Y 608.511,Z 36.895,A -85,B 0,C 180,E1 -473.437,E2 -473.437} C_VEL
LIN {X 0,Y 608.465,Z 36.692,A -85,B 0,C 180,E1 -474.149,E2 -474.149} C_VEL
LIN {X 0,Y 608.482,Z 36.685,A -85,B 0,C 180,E1 -477.207,E2 -477.207} C_VEL
LIN {X 0,Y 608.457,Z 36.692,A -85,B 0,C 180,E1 -479.969,E2 -479.969} C_VEL
LIN {X 0,Y 608.453,Z 36.689,A -85,B 0,C 180,E1 -482.88,E2 -482.88} C_VEL
LIN {X 0,Y 608.438,Z 36.69,A -85,B 0,C 180,E1 -485.278,E2 -485.278} C_VEL
LIN {X 0,Y 608.468,Z 36.691,A -85,B 0,C 180,E1 -488.24,E2 -488.24} C_VEL
LIN {X 0,Y 608.451,Z 36.691,A -85,B 0,C 180,E1 -491.341,E2 -491.341} C_VEL
LIN {X 0,Y 608.453,Z 36.69,A -85,B 0,C 180,E1 -494.263,E2 -494.263} C_VEL
LIN {X 0,Y 608.441,Z 36.691,A -85,B 0,C 180,E1 -497.039,E2 -497.039} C_VEL
LIN {X 0,Y 608.457,Z 36.694,A -85,B 0,C 180,E1 -499.697,E2 -499.697} C_VEL
LIN {X 0,Y 608.466,Z 36.686,A -85,B 0,C 180,E1 -502.253,E2 -502.253} C_VEL
LIN {X 0,Y 608.458,Z 36.695,A -85,B 0,C 180,E1 -505.094,E2 -505.094} C_VEL
LIN {X 0,Y 608.462,Z 36.687,A -85,B 0,C 180,E1 -507.905,E2 -507.905} C_VEL
LIN {X 0,Y 608.47,Z 36.686,A -85,B 0,C 180,E1 -510.22,E2 -510.22} C_VEL
LIN {X 0,Y 608.485,Z 36.692,A -85,B 0,C 180,E1 -512.792,E2 -512.792} C_VEL
LIN {X 0,Y 608.481,Z 36.684,A -85,B 0,C 180,E1 -515.848,E2 -515.848} C_VEL
LIN {X 0,Y 608.471,Z 36.689,A -85,B 0,C 180,E1 -518.308,E2 -518.308} C_VEL
LIN {X 0,Y 608.472,Z 36.686,A -85,B 0,C 180,E1 -521.285,E2 -521.285} C_VEL
LIN {X 0,Y 608.459,Z 36.689,A -85,B 0,C 180,E1 -523.906,E2 -523.906} C_VEL
LIN {X 0,Y 608.456,Z 36.693,A -85,B 0,C 180,E1 -526.643,E2 -526.643} C_VEL
LIN {X 0,Y 608.464,Z 36.686,A -85,B 0,C 180,E1 -529.35,E2 -529.35} C_VEL
LIN {X 0,Y 608.479,Z 36.693,A -85,B 0,C 180,E1 -532.033,E2 -532.033} C_VEL
LIN {X 0,Y 608.456,Z 36.689,A -85,B 0,C 180,E1 -534.698,E2 -534.698} C_VEL
LIN {X 0,Y 608.477,Z 36.687,A -85,B 0,C 180,E1 -537.352,E2 -537.352} C_VEL
LIN {X 0,Y 608.476,Z 36.692,A -85,B 0,C 180,E1 -540,E2 -540} C_VEL
LIN {X 0,Y 608.47,Z 36.686,A -85,B 0,C 180,E1 -542.648,E2 -542.648} C_VEL
LIN {X 0,Y 608.465,Z 36.691,A -85,B 0,C 180,E1 -545.302,E2 -545.302} C_VEL
LIN {X 0,Y 608.468,Z 36.689,A -85,B 0,C 180,E1 -547.967,E2 -547.967} C_VEL
LIN {X 0,Y 608.455,Z 36.693,A -85,B 0,C 180,E1 -549.447,E2 -549.447} C_VEL
LIN {X 0,Y 607.768,Z 36.776,A -85,B 0,C 180,E1 -549.999,E2 -549.999} C_VEL
LIN {X 0,Y 604.91,Z 37.132,A -85,B 0,C 180,E1 -550.896,E2 -550.896} C_VEL
LIN {X 0,Y 602.511,Z 37.434,A -85,B 0,C 180,E1 -551.618,E2 -551.618} C_VEL
LIN {X 0,Y 601.487,Z 37.556,A -85,B 0,C 180,E1 -552.174,E2 -552.174} C_VEL
LIN {X 0,Y 601.406,Z 37.566,A -85,B 0,C 180,E1 -552.363,E2 -552.363} C_VEL
LIN {X 0,Y 601.433,Z 37.567,A -85,B 0,C 180,E1 -554.897,E2 -554.897} C_VEL
LIN {X 0,Y 601.433,Z 37.57,A -85,B 0,C 180,E1 -556.986,E2 -556.986} C_VEL
LIN {X 0,Y 601.399,Z 37.567,A -85,B 0,C 180,E1 -559.81,E2 -559.81} C_VEL
LIN {X 0,Y 601.42,Z 37.569,A -85,B 0,C 180,E1 -562.605,E2 -562.605} C_VEL
LIN {X 0,Y 601.397,Z 37.576,A -85,B 0,C 180,E1 -564.879,E2 -564.879} C_VEL
LIN {X 0,Y 601.392,Z 37.569,A -85,B 0,C 180,E1 -567.357,E2 -567.357} C_VEL
LIN {X 0,Y 601.432,Z 37.566,A -85,B 0,C 180,E1 -570.148,E2 -570.148} C_VEL
LIN {X 0,Y 601.421,Z 37.57,A -85,B 0,C 180,E1 -572.715,E2 -572.715} C_VEL
LIN {X 0,Y 601.382,Z 37.57,A -85,B 0,C 180,E1 -575.11,E2 -575.11} C_VEL
LIN {X 0,Y 601.432,Z 37.563,A -85,B 0,C 180,E1 -577.419,E2 -577.419} C_VEL
LIN {X 0,Y 601.403,Z 37.573,A -85,B 0,C 180,E1 -579.996,E2 -579.996} C_VEL
LIN {X 0,Y 601.38,Z 37.571,A -85,B 0,C 180,E1 -582.673,E2 -582.673} C_VEL
LIN {X 0,Y 601.4,Z 37.569,A -85,B 0,C 180,E1 -584.532,E2 -584.532} C_VEL
LIN {X 0,Y 601.412,Z 37.568,A -85,B 0,C 180,E1 -587.409,E2 -587.409} C_VEL
LIN {X 0,Y 601.397,Z 37.573,A -85,B 0,C 180,E1 -590.004,E2 -590.004} C_VEL
LIN {X 0,Y 601.402,Z 37.566,A -85,B 0,C 180,E1 -592.622,E2 -592.622} C_VEL
LIN {X 0,Y 601.415,Z 37.567,A -85,B 0,C 180,E1 -595.068,E2 -595.068} C_VEL
LIN {X 0,Y 601.43,Z 37.573,A -85,B 0,C 180,E1 -597.484,E2 -597.484} C_VEL
LIN {X 0,Y 601.402,Z 37.57,A -85,B 0,C 180,E1 -599.856,E2 -599.856} C_VEL
LIN {X 0,Y 601.416,Z 37.652,A -85,B 0,C 180,E1 -602.615,E2 -602.615} C_VEL
LIN {X 0,Y 601.394,Z 53.033,A -85,B 0,C 180,E1 -605.455,E2 -605.455} C_VEL
LIN {X 0,Y 601.406,Z 60.853,A -85,B 0,C 180,E1 -606.885,E2 -606.885} C_VEL
LIN {X 0,Y 601.663,Z 64.331,A -85,B 0,C 180,E1 -606.941,E2 -606.941} C_VEL
LIN {X 0,Y 601.582,Z 166.866,A -85,B 0,C 180,E1 -608.182,E2 -608.182} C_VEL
LIN {X 0,Y 601.596,Z 179.941,A -85,B 0,C 180,E1 -608.476,E2 -608.476} C_VEL
LIN {X 0,Y 601.559,Z 192.53,A -85,B 0,C 180,E1 -608.894,E2 -608.894} C_VEL
LIN {X 0,Y 601.51,Z 203.854,A -85,B 0,C 180,E1 -609.401,E2 -609.401} C_VEL
LIN {X 0,Y 601.444,Z 214.592,A -85,B 0,C 180,E1 -610.014,E2 -610.014} C_VEL
LIN {X 0,Y 601.444,Z 225.713,A -85,B 0,C 180,E1 -610.813,E2 -610.813} C_VEL
LIN {X 0,Y 601.434,Z 234.72,A -85,B 0,C 180,E1 -611.609,E2 -611.609} C_VEL
LIN {X 0,Y 601.408,Z 242.933,A -85,B 0,C 180,E1 -612.488,E2 -612.488} C_VEL
LIN {X 0,Y 601.394,Z 250.448,A -85,B 0,C 180,E1 -613.477,E2 -613.477} C_VEL
LIN {X 0,Y 601.342,Z 256.206,A -85,B 0,C 180,E1 -614.407,E2 -614.407} C_VEL
LIN {X 0,Y 601.333,Z 261.35,A -85,B 0,C 180,E1 -615.447,E2 -615.447} C_VEL
LIN {X 0,Y 601.343,Z 265.286,A -85,B 0,C 180,E1 -616.482,E2 -616.482} C_VEL
LIN {X 0,Y 601.327,Z 267.295,A -85,B 0,C 180,E1 -617.17,E2 -617.17} C_VEL
LIN {X 0,Y 601.342,Z 268.872,A -85,B 0,C 180,E1 -617.856,E2 -617.856} C_VEL
LIN {X 0,Y 601.352,Z 270.538,A -85,B 0,C 180,E1 -619.025,E2 -619.025} C_VEL
LIN {X 0,Y 601.328,Z 270.973,A -85,B 0,C 180,E1 -619.903,E2 -619.903} C_VEL
LIN {X 0,Y 601.335,Z 270.872,A -85,B 0,C 180,E1 -620.583,E2 -620.583} C_VEL
LIN {X 0,Y 601.331,Z 269.393,A -85,B 0,C 180,E1 -621.938,E2 -621.938} C_VEL
LIN {X 0,Y 601.323,Z 268.061,A -85,B 0,C 180,E1 -622.613,E2 -622.613} C_VEL
LIN {X 0,Y 601.353,Z 265.908,A -85,B 0,C 180,E1 -623.41,E2 -623.41} C_VEL
LIN {X 0,Y 601.351,Z 261.383,A -85,B 0,C 180,E1 -624.635,E2 -624.635} C_VEL
LIN {X 0,Y 601.358,Z 256.421,A -85,B 0,C 180,E1 -625.643,E2 -625.643} C_VEL
LIN {X 0,Y 601.359,Z 250.206,A -85,B 0,C 180,E1 -626.65,E2 -626.65} C_VEL
LIN {X 0,Y 601.394,Z 242.468,A -85,B 0,C 180,E1 -627.656,E2 -627.656} C_VEL
LIN {X 0,Y 601.434,Z 232.838,A -85,B 0,C 180,E1 -628.661,E2 -628.661} C_VEL
LIN {X 0,Y 601.448,Z 222.903,A -85,B 0,C 180,E1 -629.498,E2 -629.498} C_VEL
LIN {X 0,Y 601.483,Z 211.723,A -85,B 0,C 180,E1 -630.251,E2 -630.251} C_VEL
LIN {X 0,Y 601.512,Z 200.817,A -85,B 0,C 180,E1 -630.837,E2 -630.837} C_VEL
LIN {X 0,Y 601.563,Z 188.746,A -85,B 0,C 180,E1 -631.339,E2 -631.339} C_VEL
LIN {X 0,Y 601.551,Z 176.128,A -85,B 0,C 180,E1 -631.716,E2 -631.716} C_VEL
LIN {X 0,Y 601.585,Z 162.844,A -85,B 0,C 180,E1 -631.967,E2 -631.967} C_VEL
LIN {X 0,Y 601.497,Z 61.923,A -85,B 0,C 180,E1 -633.182,E2 -633.182} C_VEL
LIN {X 0,Y 601.38,Z 60.75,A -85,B 0,C 180,E1 -633.224,E2 -633.224} C_VEL
LIN {X 0,Y 601.453,Z 44.398,A -85,B 0,C 180,E1 -636.223,E2 -636.223} C_VEL
LIN {X 0,Y 601.436,Z 37.564,A -85,B 0,C 180,E1 -637.512,E2 -637.512} C_VEL
LIN {X 0,Y 601.432,Z 37.564,A -85,B 0,C 180,E1 -640.095,E2 -640.095} C_VEL
LIN {X 0,Y 601.421,Z 37.571,A -85,B 0,C 180,E1 -642.828,E2 -642.828} C_VEL
LIN {X 0,Y 601.411,Z 37.565,A -85,B 0,C 180,E1 -645.592,E2 -645.592} C_VEL
LIN {X 0,Y 601.419,Z 37.574,A -85,B 0,C 180,E1 -648.392,E2 -648.392} C_VEL
LIN {X 0,Y 601.408,Z 37.565,A -85,B 0,C 180,E1 -651.24,E2 -651.24} C_VEL
LIN {X 0,Y 601.458,Z 37.568,A -85,B 0,C 180,E1 -654.141,E2 -654.141} C_VEL
LIN {X 0,Y 601.455,Z 37.559,A -85,B 0,C 180,E1 -657.111,E2 -657.111} C_VEL
LIN {X 0,Y 601.418,Z 37.565,A -85,B 0,C 180,E1 -659.393,E2 -659.393} C_VEL
LIN {X 0,Y 601.401,Z 37.573,A -85,B 0,C 180,E1 -661.727,E2 -661.727} C_VEL
LIN {X 0,Y 601.432,Z 37.568,A -85,B 0,C 180,E1 -664.119,E2 -664.119} C_VEL
LIN {X 0,Y 601.403,Z 37.566,A -85,B 0,C 180,E1 -666.583,E2 -666.583} C_VEL
LIN {X 0,Y 601.415,Z 37.567,A -85,B 0,C 180,E1 -669.127,E2 -669.127} C_VEL
LIN {X 0,Y 601.422,Z 37.571,A -85,B 0,C 180,E1 -671.766,E2 -671.766} C_VEL
LIN {X 0,Y 601.4,Z 37.566,A -85,B 0,C 180,E1 -674.533,E2 -674.533} C_VEL
LIN {X 0,Y 601.412,Z 37.575,A -85,B 0,C 180,E1 -677.41,E2 -677.41} C_VEL
LIN {X 0,Y 601.407,Z 37.566,A -85,B 0,C 180,E1 -680.005,E2 -680.005} C_VEL
LIN {X 0,Y 601.438,Z 37.563,A -85,B 0,C 180,E1 -682.618,E2 -682.618} C_VEL
LIN {X 0,Y 601.417,Z 37.574,A -85,B 0,C 180,E1 -685.068,E2 -685.068} C_VEL
LIN {X 0,Y 601.42,Z 37.567,A -85,B 0,C 180,E1 -687.484,E2 -687.484} C_VEL
LIN {X 0,Y 601.433,Z 37.562,A -85,B 0,C 180,E1 -689.852,E2 -689.852} C_VEL
LIN {X 0,Y 601.454,Z 37.569,A -85,B 0,C 180,E1 -692.889,E2 -692.889} C_VEL
LIN {X 0,Y 601.46,Z 37.559,A -85,B 0,C 180,E1 -695.86,E2 -695.86} C_VEL
LIN {X 0,Y 601.41,Z 37.573,A -85,B 0,C 180,E1 -698.761,E2 -698.761} C_VEL
LIN {X 0,Y 601.404,Z 37.566,A -85,B 0,C 180,E1 -701.608,E2 -701.608} C_VEL
LIN {X 0,Y 601.411,Z 37.575,A -85,B 0,C 180,E1 -704.409,E2 -704.409} C_VEL
LIN {X 0,Y 601.419,Z 37.564,A -85,B 0,C 180,E1 -707.172,E2 -707.172} C_VEL
LIN {X 0,Y 601.44,Z 37.566,A -85,B 0,C 180,E1 -709.905,E2 -709.905} C_VEL
LIN {X 0,Y 601.41,Z 37.568,A -85,B 0,C 180,E1 -712.615,E2 -712.615} C_VEL
LIN {X 0,Y 601.422,Z 37.564,A -85,B 0,C 180,E1 -715.308,E2 -715.308} C_VEL
LIN {X 0,Y 601.429,Z 37.572,A -85,B 0,C 180,E1 -717.991,E2 -717.991} C_VEL
LIN {X 0,Y 601.445,Z 37.561,A -85,B 0,C 180,E1 -720.67,E2 -720.67} C_VEL
LIN {X 0,Y 601.428,Z 37.567,A -85,B 0,C 180,E1 -723.35,E2 -723.35} C_VEL
LIN {X 0,Y 601.407,Z 37.569,A -85,B 0,C 180,E1 -726.037,E2 -726.037} C_VEL
LIN {X 0,Y 601.417,Z 37.565,A -85,B 0,C 180,E1 -728.738,E2 -728.738} C_VEL
LIN {X 0,Y 601.426,Z 37.573,A -85,B 0,C 180,E1 -731.458,E2 -731.458} C_VEL
LIN {X 0,Y 601.418,Z 37.564,A -85,B 0,C 180,E1 -734.206,E2 -734.206} C_VEL
LIN {X 0,Y 601.436,Z 37.568,A -85,B 0,C 180,E1 -736.986,E2 -736.986} C_VEL
LIN {X 0,Y 601.404,Z 37.567,A -85,B 0,C 180,E1 -739.81,E2 -739.81} C_VEL
LIN {X 0,Y 601.422,Z 37.567,A -85,B 0,C 180,E1 -742.605,E2 -742.605} C_VEL
LIN {X 0,Y 601.402,Z 37.575,A -85,B 0,C 180,E1 -744.879,E2 -744.879} C_VEL
LIN {X 0,Y 601.402,Z 37.569,A -85,B 0,C 180,E1 -747.359,E2 -747.359} C_VEL
LIN {X 0,Y 601.417,Z 37.566,A -85,B 0,C 180,E1 -749.393,E2 -749.393} C_VEL
LIN {X 0,Y 601.403,Z 37.566,A -85,B 0,C 180,E1 -751.727,E2 -751.727} C_VEL
LIN {X 0,Y 601.424,Z 37.566,A -85,B 0,C 180,E1 -754.119,E2 -754.119} C_VEL
LIN {X 0,Y 601.398,Z 37.576,A -85,B 0,C 180,E1 -756.584,E2 -756.584} C_VEL
LIN {X 0,Y 601.402,Z 37.567,A -85,B 0,C 180,E1 -759.127,E2 -759.127} C_VEL
LIN {X 0,Y 601.425,Z 37.565,A -85,B 0,C 180,E1 -761.765,E2 -761.765} C_VEL
LIN {X 0,Y 601.402,Z 37.571,A -85,B 0,C 180,E1 -764.532,E2 -764.532} C_VEL
LIN {X 0,Y 601.413,Z 37.565,A -85,B 0,C 180,E1 -767.409,E2 -767.409} C_VEL
LIN {X 0,Y 601.403,Z 37.576,A -85,B 0,C 180,E1 -770.004,E2 -770.004} C_VEL
LIN {X 0,Y 601.435,Z 37.563,A -85,B 0,C 180,E1 -772.618,E2 -772.618} C_VEL
LIN {X 0,Y 601.418,Z 37.565,A -85,B 0,C 180,E1 -775.068,E2 -775.068} C_VEL
LIN {X 0,Y 601.434,Z 37.567,A -85,B 0,C 180,E1 -777.484,E2 -777.484} C_VEL
LIN {X 0,Y 601.409,Z 37.573,A -85,B 0,C 180,E1 -779.855,E2 -779.855} C_VEL
LIN {X 0,Y 601.402,Z 37.569,A -85,B 0,C 180,E1 -782.131,E2 -782.131} C_VEL
LIN {X 0,Y 601.404,Z 37.567,A -85,B 0,C 180,E1 -784.381,E2 -784.381} C_VEL
LIN {X 0,Y 601.435,Z 37.736,A -85,B 0,C 180,E1 -786.385,E2 -786.385} C_VEL
LIN {X 0,Y 601.73,Z 42.012,A -85,B 0,C 180,E1 -786.966,E2 -786.966} C_VEL
LIN {X 0,Y 601.596,Z 63.848,A -85,B 0,C 180,E1 -789.841,E2 -789.841} C_VEL
LIN {X 0,Y 601.556,Z 85.684,A -85,B 0,C 180,E1 -792.667,E2 -792.667} C_VEL
LIN {X 0,Y 601.451,Z 107.521,A -85,B 0,C 180,E1 -795.45,E2 -795.45} C_VEL
LIN {X 0,Y 601.432,Z 118.353,A -85,B 0,C 180,E1 -796.818,E2 -796.818} C_VEL
LIN {X 0,Y 601.631,Z 138.804,A -85,B 0,C 180,E1 -797.069,E2 -797.069} C_VEL
LIN {X 0,Y 601.595,Z 226.938,A -85,B 0,C 180,E1 -798.139,E2 -798.139} C_VEL
LIN {X 0,Y 601.581,Z 240.212,A -85,B 0,C 180,E1 -798.438,E2 -798.438} C_VEL
LIN {X 0,Y 601.547,Z 251.896,A -85,B 0,C 180,E1 -798.825,E2 -798.825} C_VEL
LIN {X 0,Y 601.522,Z 264.63,A -85,B 0,C 180,E1 -799.396,E2 -799.396} C_VEL
LIN {X 0,Y 601.475,Z 276.197,A -85,B 0,C 180,E1 -800.076,E2 -800.076} C_VEL
LIN {X 0,Y 601.444,Z 286.594,A -85,B 0,C 180,E1 -800.839,E2 -800.839} C_VEL
LIN {X 0,Y 601.429,Z 295.111,A -85,B 0,C 180,E1 -801.601,E2 -801.601} C_VEL
LIN {X 0,Y 601.418,Z 302.959,A -85,B 0,C 180,E1 -802.446,E2 -802.446} C_VEL
LIN {X 0,Y 601.37,Z 310.225,A -85,B 0,C 180,E1 -803.398,E2 -803.398} C_VEL
LIN {X 0,Y 601.372,Z 315.866,A -85,B 0,C 180,E1 -804.299,E2 -804.299} C_VEL
LIN {X 0,Y 601.336,Z 320.95,A -85,B 0,C 180,E1 -805.307,E2 -805.307} C_VEL
LIN {X 0,Y 601.368,Z 324.896,A -85,B 0,C 180,E1 -806.315,E2 -806.315} C_VEL
LIN {X 0,Y 601.325,Z 327.809,A -85,B 0,C 180,E1 -807.32,E2 -807.32} C_VEL
LIN {X 0,Y 601.343,Z 329.202,A -85,B 0,C 180,E1 -807.991,E2 -807.991} C_VEL
LIN {X 0,Y 601.339,Z 330.784,A -85,B 0,C 180,E1 -809.33,E2 -809.33} C_VEL
LIN {X 0,Y 601.335,Z 331,A -85,B 0,C 180,E1 -810,E2 -810} C_VEL
LIN {X 0,Y 601.347,Z 330.185,A -85,B 0,C 180,E1 -811.339,E2 -811.339} C_VEL
LIN {X 0,Y 601.343,Z 329.202,A -85,B 0,C 180,E1 -812.009,E2 -812.009} C_VEL
LIN {X 0,Y 601.325,Z 327.81,A -85,B 0,C 180,E1 -812.68,E2 -812.68} C_VEL
LIN {X 0,Y 601.368,Z 324.896,A -85,B 0,C 180,E1 -813.685,E2 -813.685} C_VEL
LIN {X 0,Y 601.336,Z 320.95,A -85,B 0,C 180,E1 -814.693,E2 -814.693} C_VEL
LIN {X 0,Y 601.372,Z 314.877,A -85,B 0,C 180,E1 -815.869,E2 -815.869} C_VEL
LIN {X 0,Y 601.382,Z 308.236,A -85,B 0,C 180,E1 -816.88,E2 -816.88} C_VEL
LIN {X 0,Y 601.4,Z 299.989,A -85,B 0,C 180,E1 -817.892,E2 -817.892} C_VEL
LIN {X 0,Y 601.436,Z 291.537,A -85,B 0,C 180,E1 -818.738,E2 -818.738} C_VEL
LIN {X 0,Y 601.447,Z 281.093,A -85,B 0,C 180,E1 -819.585,E2 -819.585} C_VEL
LIN {X 0,Y 601.463,Z 270.758,A -85,B 0,C 180,E1 -820.265,E2 -820.265} C_VEL
LIN {X 0,Y 601.538,Z 258.589,A -85,B 0,C 180,E1 -820.896,E2 -820.896} C_VEL
LIN {X 0,Y 601.563,Z 246.215,A -85,B 0,C 180,E1 -821.379,E2 -821.379} C_VEL
LIN {X 0,Y 601.583,Z 233.435,A -85,B 0,C 180,E1 -821.733,E2 -821.733} C_VEL
LIN {X 0,Y 601.622,Z 221.081,A -85,B 0,C 180,E1 -821.946,E2 -821.946} C_VEL
LIN {X 0,Y 601.542,Z 119.137,A -85,B 0,C 180,E1 -823.169,E2 -823.169} C_VEL
LIN {X 0,Y 601.438,Z 118.269,A -85,B 0,C 180,E1 -823.193,E2 -823.193} C_VEL
LIN {X 0,Y 601.503,Z 95.239,A -85,B 0,C 180,E1 -826.111,E2 -826.111} C_VEL
LIN {X 0,Y 601.583,Z 75.689,A -85,B 0,C 180,E1 -828.62,E2 -828.62} C_VEL
LIN {X 0,Y 601.66,Z 54.296,A -85,B 0,C 180,E1 -831.41,E2 -831.41} C_VEL
LIN {X 0,Y 601.72,Z 39.283,A -85,B 0,C 180,E1 -833.398,E2 -833.398} C_VEL
LIN {X 0,Y 601.418,Z 37.568,A -85,B 0,C 180,E1 -833.639,E2 -833.639} C_VEL
LIN {X 0,Y 601.403,Z 37.576,A -85,B 0,C 180,E1 -836.364,E2 -836.364} C_VEL
LIN {X 0,Y 601.441,Z 37.565,A -85,B 0,C 180,E1 -838.789,E2 -838.789} C_VEL
LIN {X 0,Y 601.42,Z 37.565,A -85,B 0,C 180,E1 -841.454,E2 -841.454} C_VEL
LIN {X 0,Y 601.424,Z 37.574,A -85,B 0,C 180,E1 -844.119,E2 -844.119} C_VEL
LIN {X 0,Y 601.402,Z 37.568,A -85,B 0,C 180,E1 -846.583,E2 -846.583} C_VEL
LIN {X 0,Y 601.41,Z 37.566,A -85,B 0,C 180,E1 -849.127,E2 -849.127} C_VEL
LIN {X 0,Y 601.423,Z 37.573,A -85,B 0,C 180,E1 -851.766,E2 -851.766} C_VEL
LIN {X 0,Y 601.401,Z 37.566,A -85,B 0,C 180,E1 -854.533,E2 -854.533} C_VEL
LIN {X 0,Y 601.415,Z 37.572,A -85,B 0,C 180,E1 -857.409,E2 -857.409} C_VEL
LIN {X 0,Y 601.406,Z 37.568,A -85,B 0,C 180,E1 -860.004,E2 -860.004} C_VEL
LIN {X 0,Y 601.436,Z 37.563,A -85,B 0,C 180,E1 -862.618,E2 -862.618} C_VEL
LIN {X 0,Y 601.419,Z 37.571,A -85,B 0,C 180,E1 -865.068,E2 -865.068} C_VEL
LIN {X 0,Y 601.427,Z 37.568,A -85,B 0,C 180,E1 -867.484,E2 -867.484} C_VEL
LIN {X 0,Y 601.433,Z 37.563,A -85,B 0,C 180,E1 -869.852,E2 -869.852} C_VEL
LIN {X 0,Y 601.422,Z 37.569,A -85,B 0,C 180,E1 -872.637,E2 -872.637} C_VEL
LIN {X 0,Y 601.403,Z 37.571,A -85,B 0,C 180,E1 -875.121,E2 -875.121} C_VEL
LIN {X 0,Y 601.42,Z 37.565,A -85,B 0,C 180,E1 -878.041,E2 -878.041} C_VEL
LIN {X 0,Y 601.42,Z 37.569,A -85,B 0,C 180,E1 -880.901,E2 -880.901} C_VEL
LIN {X 0,Y 601.441,Z 37.562,A -85,B 0,C 180,E1 -883.713,E2 -883.713} C_VEL
LIN {X 0,Y 601.41,Z 37.573,A -85,B 0,C 180,E1 -886.484,E2 -886.484} C_VEL
LIN {X 0,Y 601.419,Z 37.564,A -85,B 0,C 180,E1 -889.224,E2 -889.224} C_VEL
LIN {X 0,Y 601.443,Z 37.568,A -85,B 0,C 180,E1 -891.939,E2 -891.939} C_VEL
LIN {X 0,Y 601.422,Z 37.565,A -85,B 0,C 180,E1 -894.636,E2 -894.636} C_VEL
LIN {X 0,Y 601.442,Z 37.563,A -85,B 0,C 180,E1 -897.321,E2 -897.321} C_VEL
LIN {X 0,Y 601.445,Z 37.568,A -85,B 0,C 180,E1 -900,E2 -900} C_VEL
LIN {X 0,Y 601.437,Z 37.562,A -85,B 0,C 180,E1 -902.679,E2 -902.679} C_VEL
LIN {X 0,Y 601.428,Z 37.569,A -85,B 0,C 180,E1 -905.364,E2 -905.364} C_VEL
LIN {X 0,Y 601.435,Z 37.564,A -85,B 0,C 180,E1 -908.061,E2 -908.061} C_VEL
LIN {X 0,Y 601.43,Z 37.567,A -85,B 0,C 180,E1 -911.012,E2 -911.012} C_VEL
LIN {X 0,Y 601.406,Z 37.566,A -85,B 0,C 180,E1 -912.363,E2 -912.363} C_VEL
LIN {X 0,Y 600.748,Z 37.653,A -85,B 0,C 180,E1 -912.922,E2 -912.922} C_VEL
LIN {X 0,Y 597.903,Z 38.009,A -85,B 0,C 180,E1 -913.83,E2 -913.83} C_VEL
LIN {X 0,Y 595.491,Z 38.311,A -85,B 0,C 180,E1 -914.56,E2 -914.56} C_VEL
LIN {X 0,Y 594.449,Z 38.441,A -85,B 0,C 180,E1 -915.124,E2 -915.124} C_VEL
LIN {X 0,Y 594.361,Z 38.447,A -85,B 0,C 180,E1 -915.315,E2 -915.315} C_VEL
LIN {X 0,Y 594.39,Z 38.448,A -85,B 0,C 180,E1 -917.193,E2 -917.193} C_VEL
LIN {X 0,Y 594.373,Z 38.442,A -85,B 0,C 180,E1 -920.054,E2 -920.054} C_VEL
LIN {X 0,Y 594.358,Z 38.452,A -85,B 0,C 180,E1 -922.967,E2 -922.967} C_VEL
LIN {X 0,Y 594.361,Z 38.447,A -85,B 0,C 180,E1 -925.194,E2 -925.194} C_VEL
LIN {X 0,Y 594.345,Z 38.445,A -85,B 0,C 180,E1 -927.518,E2 -927.518} C_VEL
LIN {X 0,Y 594.388,Z 38.446,A -85,B 0,C 180,E1 -930.328,E2 -930.328} C_VEL
LIN {X 0,Y 594.379,Z 38.444,A -85,B 0,C 180,E1 -932.95,E2 -932.95} C_VEL
LIN {X 0,Y 594.329,Z 38.447,A -85,B 0,C 180,E1 -935.41,E2 -935.41} C_VEL
LIN {X 0,Y 594.385,Z 38.445,A -85,B 0,C 180,E1 -937.941,E2 -937.941} C_VEL
LIN {X 0,Y 594.367,Z 38.443,A -85,B 0,C 180,E1 -940.82,E2 -940.82} C_VEL
LIN {X 0,Y 594.36,Z 38.444,A -85,B 0,C 180,E1 -943.3,E2 -943.3} C_VEL
LIN {X 0,Y 594.346,Z 38.452,A -85,B 0,C 180,E1 -946.163,E2 -946.163} C_VEL
LIN {X 0,Y 594.369,Z 38.443,A -85,B 0,C 180,E1 -948.535,E2 -948.535} C_VEL
LIN {X 0,Y 594.369,Z 38.446,A -85,B 0,C 180,E1 -951.298,E2 -951.298} C_VEL
LIN {X 0,Y 594.348,Z 38.453,A -85,B 0,C 180,E1 -953.755,E2 -953.755} C_VEL
LIN {X 0,Y 594.355,Z 38.446,A -85,B 0,C 180,E1 -956.237,E2 -956.237} C_VEL
LIN {X 0,Y 594.362,Z 38.445,A -85,B 0,C 180,E1 -958.649,E2 -958.649} C_VEL
LIN {X 0,Y 594.378,Z 38.448,A -85,B 0,C 180,E1 -961.043,E2 -961.043} C_VEL
LIN {X 0,Y 594.406,Z 38.636,A -85,B 0,C 180,E1 -962.588,E2 -962.588} C_VEL
LIN {X 0,Y 594.363,Z 53.506,A -85,B 0,C 180,E1 -965.366,E2 -965.366} C_VEL
LIN {X 0,Y 594.39,Z 60.862,A -85,B 0,C 180,E1 -966.729,E2 -966.729} C_VEL
LIN {X 0,Y 594.749,Z 65.108,A -85,B 0,C 180,E1 -966.795,E2 -966.795} C_VEL
LIN {X 0,Y 594.632,Z 167.358,A -85,B 0,C 180,E1 -968.051,E2 -968.051} C_VEL
LIN {X 0,Y 594.621,Z 181.056,A -85,B 0,C 180,E1 -968.37,E2 -968.37} C_VEL
LIN {X 0,Y 594.595,Z 194.079,A -85,B 0,C 180,E1 -968.823,E2 -968.823} C_VEL
LIN {X 0,Y 594.492,Z 206.362,A -85,B 0,C 180,E1 -969.409,E2 -969.409} C_VEL
LIN {X 0,Y 594.431,Z 218.081,A -85,B 0,C 180,E1 -970.128,E2 -970.128} C_VEL
LIN {X 0,Y 594.407,Z 228.263,A -85,B 0,C 180,E1 -970.914,E2 -970.914} C_VEL
LIN {X 0,Y 594.364,Z 237,A -85,B 0,C 180,E1 -971.739,E2 -971.739} C_VEL
LIN {X 0,Y 594.327,Z 246.189,A -85,B 0,C 180,E1 -972.805,E2 -972.805} C_VEL
LIN {X 0,Y 594.315,Z 253.45,A -85,B 0,C 180,E1 -973.865,E2 -973.865} C_VEL
LIN {X 0,Y 594.288,Z 259.191,A -85,B 0,C 180,E1 -974.92,E2 -974.92} C_VEL
LIN {X 0,Y 594.261,Z 263.313,A -85,B 0,C 180,E1 -975.876,E2 -975.876} C_VEL
LIN {X 0,Y 594.254,Z 266.98,A -85,B 0,C 180,E1 -977.014,E2 -977.014} C_VEL
LIN {X 0,Y 594.24,Z 268.617,A -85,B 0,C 180,E1 -977.709,E2 -977.709} C_VEL
LIN {X 0,Y 594.263,Z 270.52,A -85,B 0,C 180,E1 -978.99,E2 -978.99} C_VEL
LIN {X 0,Y 594.232,Z 270.946,A -85,B 0,C 180,E1 -979.781,E2 -979.781} C_VEL
LIN {X 0,Y 594.254,Z 270.908,A -85,B 0,C 180,E1 -980.47,E2 -980.47} C_VEL
LIN {X 0,Y 594.228,Z 270.466,A -85,B 0,C 180,E1 -981.156,E2 -981.156} C_VEL
LIN {X 0,Y 594.247,Z 268.313,A -85,B 0,C 180,E1 -982.525,E2 -982.525} C_VEL
LIN {X 0,Y 594.268,Z 266.006,A -85,B 0,C 180,E1 -983.419,E2 -983.419} C_VEL
LIN {X 0,Y 594.269,Z 261.881,A -85,B 0,C 180,E1 -984.571,E2 -984.571} C_VEL
LIN {X 0,Y 594.278,Z 257.055,A -85,B 0,C 180,E1 -985.591,E2 -985.591} C_VEL
LIN {X 0,Y 594.28,Z 250.988,A -85,B 0,C 180,E1 -986.61,E2 -986.61} C_VEL
LIN {X 0,Y 594.333,Z 243.465,A -85,B 0,C 180,E1 -987.628,E2 -987.628} C_VEL
LIN {X 0,Y 594.361,Z 235.815,A -85,B 0,C 180,E1 -988.476,E2 -988.476} C_VEL
LIN {X 0,Y 594.393,Z 225.468,A -85,B 0,C 180,E1 -989.407,E2 -989.407} C_VEL
LIN {X 0,Y 594.454,Z 214.979,A -85,B 0,C 180,E1 -990.169,E2 -990.169} C_VEL
LIN {X 0,Y 594.53,Z 204.869,A -85,B 0,C 180,E1 -990.762,E2 -990.762} C_VEL
LIN {X 0,Y 594.585,Z 192.944,A -85,B 0,C 180,E1 -991.312,E2 -991.312} C_VEL
LIN {X 0,Y 594.583,Z 179.799,A -85,B 0,C 180,E1 -991.757,E2 -991.757} C_VEL
LIN {X 0,Y 594.655,Z 166.567,A -85,B 0,C 180,E1 -992.053,E2 -992.053} C_VEL
LIN {X 0,Y 594.558,Z 62.442,A -85,B 0,C 180,E1 -993.331,E2 -993.331} C_VEL
LIN {X 0,Y 594.3,Z 60.719,A -85,B 0,C 180,E1 -993.39,E2 -993.39} C_VEL
LIN {X 0,Y 594.437,Z 46.061,A -85,B 0,C 180,E1 -996.108,E2 -996.108} C_VEL
LIN {X 0,Y 594.406,Z 38.441,A -85,B 0,C 180,E1 -997.559,E2 -997.559} C_VEL
LIN {X 0,Y 594.392,Z 38.443,A -85,B 0,C 180,E1 -1000.216,E2 -1000.216} C_VEL
LIN {X 0,Y 594.366,Z 38.447,A -85,B 0,C 180,E1 -1002.983,E2 -1002.983} C_VEL
LIN {X 0,Y 594.374,Z 38.444,A -85,B 0,C 180,E1 -1005.078,E2 -1005.078} C_VEL
LIN {X 0,Y 594.391,Z 38.44,A -85,B 0,C 180,E1 -1007.194,E2 -1007.194} C_VEL
LIN {X 0,Y 594.375,Z 38.446,A -85,B 0,C 180,E1 -1010.054,E2 -1010.054} C_VEL
LIN {X 0,Y 594.359,Z 38.444,A -85,B 0,C 180,E1 -1012.968,E2 -1012.968} C_VEL
LIN {X 0,Y 594.374,Z 38.442,A -85,B 0,C 180,E1 -1015.193,E2 -1015.193} C_VEL
LIN {X 0,Y 594.389,Z 38.442,A -85,B 0,C 180,E1 -1017.527,E2 -1017.527} C_VEL
LIN {X 0,Y 594.389,Z 38.445,A -85,B 0,C 180,E1 -1020.328,E2 -1020.328} C_VEL
LIN {X 0,Y 594.378,Z 38.441,A -85,B 0,C 180,E1 -1022.951,E2 -1022.951} C_VEL
LIN {X 0,Y 594.359,Z 38.447,A -85,B 0,C 180,E1 -1025.409,E2 -1025.409} C_VEL
LIN {X 0,Y 594.386,Z 38.447,A -85,B 0,C 180,E1 -1027.941,E2 -1027.941} C_VEL
LIN {X 0,Y 594.376,Z 38.442,A -85,B 0,C 180,E1 -1030.822,E2 -1030.822} C_VEL
LIN {X 0,Y 594.369,Z 38.448,A -85,B 0,C 180,E1 -1033.3,E2 -1033.3} C_VEL
LIN {X 0,Y 594.363,Z 38.444,A -85,B 0,C 180,E1 -1036.162,E2 -1036.162} C_VEL
LIN {X 0,Y 594.381,Z 38.441,A -85,B 0,C 180,E1 -1038.536,E2 -1038.536} C_VEL
LIN {X 0,Y 594.385,Z 38.45,A -85,B 0,C 180,E1 -1041.296,E2 -1041.296} C_VEL
LIN {X 0,Y 594.355,Z 38.446,A -85,B 0,C 180,E1 -1043.756,E2 -1043.756} C_VEL
LIN {X 0,Y 594.379,Z 38.441,A -85,B 0,C 180,E1 -1046.239,E2 -1046.239} C_VEL
LIN {X 0,Y 594.373,Z 38.446,A -85,B 0,C 180,E1 -1048.65,E2 -1048.65} C_VEL
LIN {X 0,Y 594.385,Z 38.448,A -85,B 0,C 180,E1 -1051.043,E2 -1051.043} C_VEL
LIN {X 0,Y 594.386,Z 38.443,A -85,B 0,C 180,E1 -1053.301,E2 -1053.301} C_VEL
LIN {X 0,Y 594.391,Z 38.443,A -85,B 0,C 180,E1 -1056.296,E2 -1056.296} C_VEL
LIN {X 0,Y 594.403,Z 38.439,A -85,B 0,C 180,E1 -1059.224,E2 -1059.224} C_VEL
LIN {X 0,Y 594.348,Z 38.449,A -85,B 0,C 180,E1 -1062.095,E2 -1062.095} C_VEL
LIN {X 0,Y 594.366,Z 38.449,A -85,B 0,C 180,E1 -1064.219,E2 -1064.219} C_VEL
LIN {X 0,Y 594.382,Z 38.451,A -85,B 0,C 180,E1 -1066.321,E2 -1066.321} C_VEL
LIN {X 0,Y 594.378,Z 38.441,A -85,B 0,C 180,E1 -1069.095,E2 -1069.095} C_VEL
LIN {X 0,Y 594.389,Z 38.445,A -85,B 0,C 180,E1 -1071.843,E2 -1071.843} C_VEL
LIN {X 0,Y 594.388,Z 38.442,A -85,B 0,C 180,E1 -1074.572,E2 -1074.572} C_VEL
LIN {X 0,Y 594.408,Z 38.439,A -85,B 0,C 180,E1 -1077.289,E2 -1077.289} C_VEL
LIN {X 0,Y 594.416,Z 38.444,A -85,B 0,C 180,E1 -1080,E2 -1080} C_VEL
LIN {X 0,Y 594.404,Z 38.438,A -85,B 0,C 180,E1 -1082.711,E2 -1082.711} C_VEL
LIN {X 0,Y 594.391,Z 38.446,A -85,B 0,C 180,E1 -1085.428,E2 -1085.428} C_VEL
LIN {X 0,Y 594.385,Z 38.442,A -85,B 0,C 180,E1 -1088.157,E2 -1088.157} C_VEL
LIN {X 0,Y 594.395,Z 38.443,A -85,B 0,C 180,E1 -1091.073,E2 -1091.073} C_VEL
LIN {X 0,Y 594.374,Z 38.446,A -85,B 0,C 180,E1 -1093.679,E2 -1093.679} C_VEL
LIN {X 0,Y 594.399,Z 38.441,A -85,B 0,C 180,E1 -1096.719,E2 -1096.719} C_VEL
LIN {X 0,Y 594.37,Z 38.449,A -85,B 0,C 180,E1 -1099.334,E2 -1099.334} C_VEL
LIN {X 0,Y 594.366,Z 38.446,A -85,B 0,C 180,E1 -1101.503,E2 -1101.503} C_VEL
LIN {X 0,Y 594.395,Z 38.441,A -85,B 0,C 180,E1 -1104.446,E2 -1104.446} C_VEL
LIN {X 0,Y 594.381,Z 38.442,A -85,B 0,C 180,E1 -1107.461,E2 -1107.461} C_VEL
LIN {X 0,Y 594.391,Z 38.443,A -85,B 0,C 180,E1 -1110.328,E2 -1110.328} C_VEL
LIN {X 0,Y 594.381,Z 38.446,A -85,B 0,C 180,E1 -1112.95,E2 -1112.95} C_VEL
LIN {X 0,Y 594.352,Z 38.445,A -85,B 0,C 180,E1 -1115.409,E2 -1115.409} C_VEL
LIN {X 0,Y 594.386,Z 38.442,A -85,B 0,C 180,E1 -1117.941,E2 -1117.941} C_VEL
LIN {X 0,Y 594.373,Z 38.445,A -85,B 0,C 180,E1 -1120.821,E2 -1120.821} C_VEL
LIN {X 0,Y 594.37,Z 38.442,A -85,B 0,C 180,E1 -1123.299,E2 -1123.299} C_VEL
LIN {X 0,Y 594.349,Z 38.455,A -85,B 0,C 180,E1 -1126.163,E2 -1126.163} C_VEL
LIN {X 0,Y 594.376,Z 38.445,A -85,B 0,C 180,E1 -1128.535,E2 -1128.535} C_VEL
LIN {X 0,Y 594.375,Z 38.442,A -85,B 0,C 180,E1 -1131.297,E2 -1131.297} C_VEL
LIN {X 0,Y 594.354,Z 38.451,A -85,B 0,C 180,E1 -1133.755,E2 -1133.755} C_VEL
LIN {X 0,Y 594.368,Z 38.446,A -85,B 0,C 180,E1 -1136.238,E2 -1136.238} C_VEL
LIN {X 0,Y 594.37,Z 38.442,A -85,B 0,C 180,E1 -1138.649,E2 -1138.649} C_VEL
LIN {X 0,Y 594.387,Z 38.442,A -85,B 0,C 180,E1 -1141.042,E2 -1141.042} C_VEL
LIN {X 0,Y 594.377,Z 38.445,A -85,B 0,C 180,E1 -1143.98,E2 -1143.98} C_VEL
LIN {X 0,Y 594.406,Z 38.62,A -85,B 0,C 180,E1 -1146.25,E2 -1146.25} C_VEL
LIN {X 0,Y 594.812,Z 43.185,A -85,B 0,C 180,E1 -1146.867,E2 -1146.867} C_VEL
LIN {X 0,Y 594.693,Z 63.848,A -85,B 0,C 180,E1 -1149.596,E2 -1149.596} C_VEL
LIN {X 0,Y 594.598,Z 85.684,A -85,B 0,C 180,E1 -1152.458,E2 -1152.458} C_VEL
LIN {X 0,Y 594.443,Z 107.521,A -85,B 0,C 180,E1 -1155.274,E2 -1155.274} C_VEL
LIN {X 0,Y 594.435,Z 118.353,A -85,B 0,C 180,E1 -1156.66,E2 -1156.66} C_VEL
LIN {X 0,Y 594.741,Z 124.494,A -85,B 0,C 180,E1 -1156.743,E2 -1156.743} C_VEL
LIN {X 0,Y 594.664,Z 226.938,A -85,B 0,C 180,E1 -1157.999,E2 -1157.999} C_VEL
LIN {X 0,Y 594.624,Z 240.213,A -85,B 0,C 180,E1 -1158.301,E2 -1158.301} C_VEL
LIN {X 0,Y 594.592,Z 253.266,A -85,B 0,C 180,E1 -1158.745,E2 -1158.745} C_VEL
LIN {X 0,Y 594.536,Z 264.628,A -85,B 0,C 180,E1 -1159.27,E2 -1159.27} C_VEL
LIN {X 0,Y 594.471,Z 276.199,A -85,B 0,C 180,E1 -1159.957,E2 -1159.957} C_VEL
LIN {X 0,Y 594.414,Z 286.596,A -85,B 0,C 180,E1 -1160.729,E2 -1160.729} C_VEL
LIN {X 0,Y 594.383,Z 295.111,A -85,B 0,C 180,E1 -1161.5,E2 -1161.5} C_VEL
LIN {X 0,Y 594.347,Z 302.959,A -85,B 0,C 180,E1 -1162.355,E2 -1162.355} C_VEL
LIN {X 0,Y 594.283,Z 310.813,A -85,B 0,C 180,E1 -1163.408,E2 -1163.408} C_VEL
LIN {X 0,Y 594.289,Z 317.68,A -85,B 0,C 180,E1 -1164.571,E2 -1164.571} C_VEL
LIN {X 0,Y 594.27,Z 322.371,A -85,B 0,C 180,E1 -1165.591,E2 -1165.591} C_VEL
LIN {X 0,Y 594.267,Z 325.956,A -85,B 0,C 180,E1 -1166.61,E2 -1166.61} C_VEL
LIN {X 0,Y 594.226,Z 327.808,A -85,B 0,C 180,E1 -1167.288,E2 -1167.288} C_VEL
LIN {X 0,Y 594.242,Z 329.2,A -85,B 0,C 180,E1 -1167.967,E2 -1167.967} C_VEL
LIN {X 0,Y 594.239,Z 330.784,A -85,B 0,C 180,E1 -1169.322,E2 -1169.322} C_VEL
LIN {X 0,Y 594.236,Z 331,A -85,B 0,C 180,E1 -1170,E2 -1170} C_VEL
LIN {X 0,Y 594.247,Z 330.185,A -85,B 0,C 180,E1 -1171.355,E2 -1171.355} C_VEL
LIN {X 0,Y 594.242,Z 329.201,A -85,B 0,C 180,E1 -1172.033,E2 -1172.033} C_VEL
LIN {X 0,Y 594.226,Z 327.81,A -85,B 0,C 180,E1 -1172.712,E2 -1172.712} C_VEL
LIN {X 0,Y 594.289,Z 324.896,A -85,B 0,C 180,E1 -1173.729,E2 -1173.729} C_VEL
LIN {X 0,Y 594.241,Z 320.949,A -85,B 0,C 180,E1 -1174.749,E2 -1174.749} C_VEL
LIN {X 0,Y 594.305,Z 314.877,A -85,B 0,C 180,E1 -1175.939,E2 -1175.939} C_VEL
LIN {X 0,Y 594.308,Z 308.237,A -85,B 0,C 180,E1 -1176.962,E2 -1176.962} C_VEL
LIN {X 0,Y 594.359,Z 299.99,A -85,B 0,C 180,E1 -1177.986,E2 -1177.986} C_VEL
LIN {X 0,Y 594.382,Z 291.537,A -85,B 0,C 180,E1 -1178.842,E2 -1178.842} C_VEL
LIN {X 0,Y 594.428,Z 281.095,A -85,B 0,C 180,E1 -1179.699,E2 -1179.699} C_VEL
LIN {X 0,Y 594.471,Z 270.757,A -85,B 0,C 180,E1 -1180.387,E2 -1180.387} C_VEL
LIN {X 0,Y 594.558,Z 259.723,A -85,B 0,C 180,E1 -1180.973,E2 -1180.973} C_VEL
LIN {X 0,Y 594.584,Z 247.71,A -85,B 0,C 180,E1 -1181.464,E2 -1181.464} C_VEL
LIN {X 0,Y 594.633,Z 234.348,A -85,B 0,C 180,E1 -1181.85,E2 -1181.85} C_VEL
LIN {X 0,Y 594.695,Z 221.081,A -85,B 0,C 180,E1 -1182.087,E2 -1182.087} C_VEL
LIN {X 0,Y 594.635,Z 119.808,A -85,B 0,C 180,E1 -1183.317,E2 -1183.317} C_VEL
LIN {X 0,Y 594.442,Z 118.269,A -85,B 0,C 180,E1 -1183.351,E2 -1183.351} C_VEL
LIN {X 0,Y 594.524,Z 95.239,A -85,B 0,C 180,E1 -1186.305,E2 -1186.305} C_VEL
LIN {X 0,Y 594.6,Z 75.491,A -85,B 0,C 180,E1 -1188.873,E2 -1188.873} C_VEL
LIN {X 0,Y 594.741,Z 55.661,A -85,B 0,C 180,E1 -1191.489,E2 -1191.489} C_VEL
LIN {X 0,Y 594.728,Z 40.348,A -85,B 0,C 180,E1 -1193.505,E2 -1193.505} C_VEL
LIN {X 0,Y 594.387,Z 38.445,A -85,B 0,C 180,E1 -1193.797,E2 -1193.797} C_VEL
LIN {X 0,Y 594.388,Z 38.446,A -85,B 0,C 180,E1 -1196.7,E2 -1196.7} C_VEL
LIN {X 0,Y 594.383,Z 38.442,A -85,B 0,C 180,E1 -1198.999,E2 -1198.999} C_VEL
LIN {X 0,Y 594.378,Z 38.443,A -85,B 0,C 180,E1 -1201.642,E2 -1201.642} C_VEL
LIN {X 0,Y 594.384,Z 38.443,A -85,B 0,C 180,E1 -1204.58,E2 -1204.58} C_VEL
LIN {X 0,Y 594.391,Z 38.444,A -85,B 0,C 180,E1 -1207.608,E2 -1207.608} C_VEL
LIN {X 0,Y 594.37,Z 38.443,A -85,B 0,C 180,E1 -1210.567,E2 -1210.567} C_VEL
LIN {X 0,Y 594.368,Z 38.446,A -85,B 0,C 180,E1 -1213.3,E2 -1213.3} C_VEL
LIN {X 0,Y 594.364,Z 38.445,A -85,B 0,C 180,E1 -1216.161,E2 -1216.161} C_VEL
LIN {X 0,Y 594.38,Z 38.441,A -85,B 0,C 180,E1 -1218.536,E2 -1218.536} C_VEL
LIN {X 0,Y 594.384,Z 38.448,A -85,B 0,C 180,E1 -1221.296,E2 -1221.296} C_VEL
LIN {X 0,Y 594.356,Z 38.447,A -85,B 0,C 180,E1 -1223.756,E2 -1223.756} C_VEL
LIN {X 0,Y 594.368,Z 38.442,A -85,B 0,C 180,E1 -1226.238,E2 -1226.238} C_VEL
LIN {X 0,Y 594.373,Z 38.445,A -85,B 0,C 180,E1 -1228.65,E2 -1228.65} C_VEL
LIN {X 0,Y 594.386,Z 38.45,A -85,B 0,C 180,E1 -1231.043,E2 -1231.043} C_VEL
LIN {X 0,Y 594.388,Z 38.443,A -85,B 0,C 180,E1 -1233.3,E2 -1233.3} C_VEL
LIN {X 0,Y 594.379,Z 38.444,A -85,B 0,C 180,E1 -1236.295,E2 -1236.295} C_VEL
LIN {X 0,Y 594.404,Z 38.44,A -85,B 0,C 180,E1 -1239.224,E2 -1239.224} C_VEL
LIN {X 0,Y 594.348,Z 38.448,A -85,B 0,C 180,E1 -1242.095,E2 -1242.095} C_VEL
LIN {X 0,Y 594.366,Z 38.448,A -85,B 0,C 180,E1 -1244.219,E2 -1244.219} C_VEL
LIN {X 0,Y 594.379,Z 38.45,A -85,B 0,C 180,E1 -1246.321,E2 -1246.321} C_VEL
LIN {X 0,Y 594.378,Z 38.441,A -85,B 0,C 180,E1 -1249.095,E2 -1249.095} C_VEL
LIN {X 0,Y 594.417,Z 38.441,A -85,B 0,C 180,E1 -1251.843,E2 -1251.843} C_VEL
LIN {X 0,Y 594.388,Z 38.442,A -85,B 0,C 180,E1 -1254.572,E2 -1254.572} C_VEL
LIN {X 0,Y 594.408,Z 38.439,A -85,B 0,C 180,E1 -1257.289,E2 -1257.289} C_VEL
LIN {X 0,Y 594.415,Z 38.444,A -85,B 0,C 180,E1 -1260,E2 -1260} C_VEL
LIN {X 0,Y 594.404,Z 38.438,A -85,B 0,C 180,E1 -1262.711,E2 -1262.711} C_VEL
LIN {X 0,Y 594.391,Z 38.446,A -85,B 0,C 180,E1 -1265.428,E2 -1265.428} C_VEL
LIN {X 0,Y 594.382,Z 38.441,A -85,B 0,C 180,E1 -1268.157,E2 -1268.157} C_VEL
LIN {X 0,Y 594.394,Z 38.444,A -85,B 0,C 180,E1 -1271.073,E2 -1271.073} C_VEL
LIN {X 0,Y 594.374,Z 38.445,A -85,B 0,C 180,E1 -1273.679,E2 -1273.679} C_VEL
LIN {X 0,Y 594.361,Z 38.447,A -85,B 0,C 180,E1 -1275.315,E2 -1275.315} C_VEL
LIN {X 0,Y 593.682,Z 38.53,A -85,B 0,C 180,E1 -1275.88,E2 -1275.88} C_VEL
LIN {X 0,Y 590.81,Z 38.89,A -85,B 0,C 180,E1 -1276.798,E2 -1276.798} C_VEL
LIN {X 0,Y 588.399,Z 39.189,A -85,B 0,C 180,E1 -1277.537,E2 -1277.537} C_VEL
LIN {X 0,Y 587.379,Z 39.313,A -85,B 0,C 180,E1 -1278.107,E2 -1278.107} C_VEL
LIN {X 0,Y 587.304,Z 39.323,A -85,B 0,C 180,E1 -1278.3,E2 -1278.3} C_VEL
LIN {X 0,Y 587.335,Z 39.327,A -85,B 0,C 180,E1 -1281.037,E2 -1281.037} C_VEL
LIN {X 0,Y 587.315,Z 39.325,A -85,B 0,C 180,E1 -1283.259,E2 -1283.259} C_VEL
LIN {X 0,Y 587.323,Z 39.321,A -85,B 0,C 180,E1 -1285.517,E2 -1285.517} C_VEL
LIN {X 0,Y 587.307,Z 39.322,A -85,B 0,C 180,E1 -1287.82,E2 -1287.82} C_VEL
LIN {X 0,Y 587.337,Z 39.327,A -85,B 0,C 180,E1 -1290.509,E2 -1290.509} C_VEL
LIN {X 0,Y 587.329,Z 39.319,A -85,B 0,C 180,E1 -1293.397,E2 -1293.397} C_VEL
LIN {X 0,Y 587.285,Z 39.328,A -85,B 0,C 180,E1 -1295.901,E2 -1295.901} C_VEL
LIN {X 0,Y 587.322,Z 39.326,A -85,B 0,C 180,E1 -1298.48,E2 -1298.48} C_VEL
LIN {X 0,Y 587.334,Z 39.318,A -85,B 0,C 180,E1 -1301.157,E2 -1301.157} C_VEL
LIN {X 0,Y 587.315,Z 39.33,A -85,B 0,C 180,E1 -1304.112,E2 -1304.112} C_VEL
LIN {X 0,Y 587.305,Z 39.323,A -85,B 0,C 180,E1 -1306.992,E2 -1306.992} C_VEL
LIN {X 0,Y 587.308,Z 39.332,A -85,B 0,C 180,E1 -1309.745,E2 -1309.745} C_VEL
LIN {X 0,Y 587.32,Z 39.322,A -85,B 0,C 180,E1 -1312.39,E2 -1312.39} C_VEL
LIN {X 0,Y 587.339,Z 39.327,A -85,B 0,C 180,E1 -1315.654,E2 -1315.654} C_VEL
LIN {X 0,Y 587.333,Z 39.321,A -85,B 0,C 180,E1 -1318.23,E2 -1318.23} C_VEL
LIN {X 0,Y 587.343,Z 39.322,A -85,B 0,C 180,E1 -1320.868,E2 -1320.868} C_VEL
LIN {X 0,Y 587.372,Z 39.427,A -85,B 0,C 180,E1 -1322.523,E2 -1322.523} C_VEL
LIN {X 0,Y 587.319,Z 53.791,A -85,B 0,C 180,E1 -1325.24,E2 -1325.24} C_VEL
LIN {X 0,Y 587.347,Z 60.868,A -85,B 0,C 180,E1 -1326.567,E2 -1326.567} C_VEL
LIN {X 0,Y 587.846,Z 66.779,A -85,B 0,C 180,E1 -1326.657,E2 -1326.657} C_VEL
LIN {X 0,Y 587.722,Z 166.672,A -85,B 0,C 180,E1 -1327.895,E2 -1327.895} C_VEL
LIN {X 0,Y 587.654,Z 179.772,A -85,B 0,C 180,E1 -1328.192,E2 -1328.192} C_VEL
LIN {X 0,Y 587.608,Z 192.003,A -85,B 0,C 180,E1 -1328.606,E2 -1328.606} C_VEL
LIN {X 0,Y 587.536,Z 204.029,A -85,B 0,C 180,E1 -1329.153,E2 -1329.153} C_VEL
LIN {X 0,Y 587.447,Z 214.86,A -85,B 0,C 180,E1 -1329.791,E2 -1329.791} C_VEL
LIN {X 0,Y 587.389,Z 225.62,A -85,B 0,C 180,E1 -1330.582,E2 -1330.582} C_VEL
LIN {X 0,Y 587.35,Z 235.814,A -85,B 0,C 180,E1 -1331.513,E2 -1331.513} C_VEL
LIN {X 0,Y 587.263,Z 245.203,A -85,B 0,C 180,E1 -1332.591,E2 -1332.591} C_VEL
LIN {X 0,Y 587.195,Z 252.695,A -85,B 0,C 180,E1 -1333.664,E2 -1333.664} C_VEL
LIN {X 0,Y 587.187,Z 258.607,A -85,B 0,C 180,E1 -1334.733,E2 -1334.733} C_VEL
LIN {X 0,Y 587.163,Z 263.287,A -85,B 0,C 180,E1 -1335.818,E2 -1335.818} C_VEL
LIN {X 0,Y 587.162,Z 266.66,A -85,B 0,C 180,E1 -1336.855,E2 -1336.855} C_VEL
LIN {X 0,Y 587.162,Z 268.363,A -85,B 0,C 180,E1 -1337.558,E2 -1337.558} C_VEL
LIN {X 0,Y 587.154,Z 269.64,A -85,B 0,C 180,E1 -1338.259,E2 -1338.259} C_VEL
LIN {X 0,Y 587.164,Z 270.504,A -85,B 0,C 180,E1 -1338.959,E2 -1338.959} C_VEL
LIN {X 0,Y 587.15,Z 270.936,A -85,B 0,C 180,E1 -1340.353,E2 -1340.353} C_VEL
LIN {X 0,Y 587.127,Z 270.566,A -85,B 0,C 180,E1 -1341.048,E2 -1341.048} C_VEL
LIN {X 0,Y 587.137,Z 269.782,A -85,B 0,C 180,E1 -1341.742,E2 -1341.742} C_VEL
LIN {X 0,Y 587.145,Z 268.566,A -85,B 0,C 180,E1 -1342.434,E2 -1342.434} C_VEL
LIN {X 0,Y 587.194,Z 266.134,A -85,B 0,C 180,E1 -1343.418,E2 -1343.418} C_VEL
LIN {X 0,Y 587.189,Z 262.378,A -85,B 0,C 180,E1 -1344.505,E2 -1344.505} C_VEL
LIN {X 0,Y 587.198,Z 257.687,A -85,B 0,C 180,E1 -1345.538,E2 -1345.538} C_VEL
LIN {X 0,Y 587.219,Z 250.653,A -85,B 0,C 180,E1 -1346.741,E2 -1346.741} C_VEL
LIN {X 0,Y 587.256,Z 243.056,A -85,B 0,C 180,E1 -1347.771,E2 -1347.771} C_VEL
LIN {X 0,Y 587.346,Z 233.544,A -85,B 0,C 180,E1 -1348.8,E2 -1348.8} C_VEL
LIN {X 0,Y 587.389,Z 223.78,A -85,B 0,C 180,E1 -1349.657,E2 -1349.657} C_VEL
LIN {X 0,Y 587.45,Z 212.848,A -85,B 0,C 180,E1 -1350.428,E2 -1350.428} C_VEL
LIN {X 0,Y 587.544,Z 200.466,A -85,B 0,C 180,E1 -1351.114,E2 -1351.114} C_VEL
LIN {X 0,Y 587.635,Z 188.266,A -85,B 0,C 180,E1 -1351.628,E2 -1351.628} C_VEL
LIN {X 0,Y 587.651,Z 175.392,A -85,B 0,C 180,E1 -1352.013,E2 -1352.013} C_VEL
LIN {X 0,Y 587.741,Z 161.582,A -85,B 0,C 180,E1 -1352.27,E2 -1352.27} C_VEL
LIN {X 0,Y 587.672,Z 63.308,A -85,B 0,C 180,E1 -1353.479,E2 -1353.479} C_VEL
LIN {X 0,Y 587.277,Z 60.797,A -85,B 0,C 180,E1 -1353.538,E2 -1353.538} C_VEL
LIN {X 0,Y 587.406,Z 46.717,A -85,B 0,C 180,E1 -1356.182,E2 -1356.182} C_VEL
LIN {X 0,Y 587.373,Z 39.317,A -85,B 0,C 180,E1 -1357.606,E2 -1357.606} C_VEL
LIN {X 0,Y 587.342,Z 39.323,A -85,B 0,C 180,E1 -1360.34,E2 -1360.34} C_VEL
LIN {X 0,Y 587.316,Z 39.323,A -85,B 0,C 180,E1 -1363.142,E2 -1363.142} C_VEL
LIN {X 0,Y 587.331,Z 39.32,A -85,B 0,C 180,E1 -1365.263,E2 -1365.263} C_VEL
LIN {X 0,Y 587.351,Z 39.316,A -85,B 0,C 180,E1 -1367.406,E2 -1367.406} C_VEL
LIN {X 0,Y 587.33,Z 39.328,A -85,B 0,C 180,E1 -1370.305,E2 -1370.305} C_VEL
LIN {X 0,Y 587.316,Z 39.321,A -85,B 0,C 180,E1 -1373.259,E2 -1373.259} C_VEL
LIN {X 0,Y 587.333,Z 39.32,A -85,B 0,C 180,E1 -1375.517,E2 -1375.517} C_VEL
LIN {X 0,Y 587.351,Z 39.322,A -85,B 0,C 180,E1 -1377.818,E2 -1377.818} C_VEL
LIN {X 0,Y 587.339,Z 39.32,A -85,B 0,C 180,E1 -1380.51,E2 -1380.51} C_VEL
LIN {X 0,Y 587.335,Z 39.321,A -85,B 0,C 180,E1 -1383.397,E2 -1383.397} C_VEL
LIN {X 0,Y 587.297,Z 39.332,A -85,B 0,C 180,E1 -1385.9,E2 -1385.9} C_VEL
LIN {X 0,Y 587.33,Z 39.32,A -85,B 0,C 180,E1 -1388.48,E2 -1388.48} C_VEL
LIN {X 0,Y 587.337,Z 39.321,A -85,B 0,C 180,E1 -1391.157,E2 -1391.157} C_VEL
LIN {X 0,Y 587.315,Z 39.323,A -85,B 0,C 180,E1 -1394.112,E2 -1394.112} C_VEL
LIN {X 0,Y 587.316,Z 39.324,A -85,B 0,C 180,E1 -1396.994,E2 -1396.994} C_VEL
LIN {X 0,Y 587.314,Z 39.324,A -85,B 0,C 180,E1 -1399.746,E2 -1399.746} C_VEL
LIN {X 0,Y 587.347,Z 39.317,A -85,B 0,C 180,E1 -1402.392,E2 -1402.392} C_VEL
LIN {X 0,Y 587.353,Z 39.318,A -85,B 0,C 180,E1 -1405.652,E2 -1405.652} C_VEL
LIN {X 0,Y 587.341,Z 39.318,A -85,B 0,C 180,E1 -1408.231,E2 -1408.231} C_VEL
LIN {X 0,Y 587.353,Z 39.326,A -85,B 0,C 180,E1 -1410.867,E2 -1410.867} C_VEL
LIN {X 0,Y 587.341,Z 39.318,A -85,B 0,C 180,E1 -1413.722,E2 -1413.722} C_VEL
LIN {X 0,Y 587.34,Z 39.319,A -85,B 0,C 180,E1 -1415.994,E2 -1415.994} C_VEL
LIN {X 0,Y 587.325,Z 39.323,A -85,B 0,C 180,E1 -1418.226,E2 -1418.226} C_VEL
LIN {X 0,Y 587.35,Z 39.318,A -85,B 0,C 180,E1 -1421.151,E2 -1421.151} C_VEL
LIN {X 0,Y 587.322,Z 39.324,A -85,B 0,C 180,E1 -1424.025,E2 -1424.025} C_VEL
LIN {X 0,Y 587.361,Z 39.322,A -85,B 0,C 180,E1 -1426.154,E2 -1426.154} C_VEL
LIN {X 0,Y 587.345,Z 39.318,A -85,B 0,C 180,E1 -1428.963,E2 -1428.963} C_VEL
LIN {X 0,Y 587.348,Z 39.32,A -85,B 0,C 180,E1 -1431.745,E2 -1431.745} C_VEL
LIN {X 0,Y 587.355,Z 39.319,A -85,B 0,C 180,E1 -1434.507,E2 -1434.507} C_VEL
LIN {X 0,Y 587.374,Z 39.315,A -85,B 0,C 180,E1 -1437.257,E2 -1437.257} C_VEL
LIN {X 0,Y 587.385,Z 39.32,A -85,B 0,C 180,E1 -1440,E2 -1440} C_VEL
LIN {X 0,Y 587.371,Z 39.314,A -85,B 0,C 180,E1 -1442.743,E2 -1442.743} C_VEL
LIN {X 0,Y 587.356,Z 39.323,A -85,B 0,C 180,E1 -1445.493,E2 -1445.493} C_VEL
LIN {X 0,Y 587.345,Z 39.318,A -85,B 0,C 180,E1 -1448.256,E2 -1448.256} C_VEL
LIN {X 0,Y 587.355,Z 39.321,A -85,B 0,C 180,E1 -1451.134,E2 -1451.134} C_VEL
LIN {X 0,Y 587.363,Z 39.315,A -85,B 0,C 180,E1 -1454.257,E2 -1454.257} C_VEL
LIN {X 0,Y 587.352,Z 39.323,A -85,B 0,C 180,E1 -1457.406,E2 -1457.406} C_VEL
LIN {X 0,Y 587.331,Z 39.319,A -85,B 0,C 180,E1 -1460.305,E2 -1460.305} C_VEL
LIN {X 0,Y 587.317,Z 39.327,A -85,B 0,C 180,E1 -1463.259,E2 -1463.259} C_VEL
LIN {X 0,Y 587.327,Z 39.321,A -85,B 0,C 180,E1 -1465.517,E2 -1465.517} C_VEL
LIN {X 0,Y 587.312,Z 39.321,A -85,B 0,C 180,E1 -1467.82,E2 -1467.82} C_VEL
LIN {X 0,Y 587.34,Z 39.324,A -85,B 0,C 180,E1 -1470.509,E2 -1470.509} C_VEL
LIN {X 0,Y 587.332,Z 39.319,A -85,B 0,C 180,E1 -1473.397,E2 -1473.397} C_VEL
LIN {X 0,Y 587.295,Z 39.325,A -85,B 0,C 180,E1 -1475.9,E2 -1475.9} C_VEL
LIN {X 0,Y 587.325,Z 39.33,A -85,B 0,C 180,E1 -1478.48,E2 -1478.48} C_VEL
LIN {X 0,Y 587.337,Z 39.319,A -85,B 0,C 180,E1 -1481.157,E2 -1481.157} C_VEL
LIN {X 0,Y 587.316,Z 39.328,A -85,B 0,C 180,E1 -1484.112,E2 -1484.112} C_VEL
LIN {X 0,Y 587.308,Z 39.322,A -85,B 0,C 180,E1 -1486.992,E2 -1486.992} C_VEL
LIN {X 0,Y 587.314,Z 39.326,A -85,B 0,C 180,E1 -1489.745,E2 -1489.745} C_VEL
LIN {X 0,Y 587.345,Z 39.321,A -85,B 0,C 180,E1 -1492.392,E2 -1492.392} C_VEL
LIN {X 0,Y 587.348,Z 39.324,A -85,B 0,C 180,E1 -1495.653,E2 -1495.653} C_VEL
LIN {X 0,Y 587.342,Z 39.32,A -85,B 0,C 180,E1 -1498.231,E2 -1498.231} C_VEL
LIN {X 0,Y 587.351,Z 39.318,A -85,B 0,C 180,E1 -1500.867,E2 -1500.867} C_VEL
LIN {X 0,Y 587.34,Z 39.325,A -85,B 0,C 180,E1 -1503.824,E2 -1503.824} C_VEL
LIN {X 0,Y 587.363,Z 39.483,A -85,B 0,C 180,E1 -1506.112,E2 -1506.112} C_VEL
LIN {X 0,Y 587.884,Z 44.235,A -85,B 0,C 180,E1 -1506.765,E2 -1506.765} C_VEL
LIN {X 0,Y 587.749,Z 66.572,A -85,B 0,C 180,E1 -1509.71,E2 -1509.71} C_VEL
LIN {X 0,Y 587.634,Z 89.624,A -85,B 0,C 180,E1 -1512.762,E2 -1512.762} C_VEL
LIN {X 0,Y 587.457,Z 111.762,A -85,B 0,C 180,E1 -1515.645,E2 -1515.645} C_VEL
LIN {X 0,Y 587.4,Z 118.353,A -85,B 0,C 180,E1 -1516.497,E2 -1516.497} C_VEL
LIN {X 0,Y 587.847,Z 122.705,A -85,B 0,C 180,E1 -1516.562,E2 -1516.562} C_VEL
LIN {X 0,Y 587.725,Z 226.938,A -85,B 0,C 180,E1 -1517.855,E2 -1517.855} C_VEL
LIN {X 0,Y 587.671,Z 240.214,A -85,B 0,C 180,E1 -1518.16,E2 -1518.16} C_VEL
LIN {X 0,Y 587.615,Z 252.638,A -85,B 0,C 180,E1 -1518.585,E2 -1518.585} C_VEL
LIN {X 0,Y 587.558,Z 264.626,A -85,B 0,C 180,E1 -1519.141,E2 -1519.141} C_VEL
LIN {X 0,Y 587.458,Z 276.2,A -85,B 0,C 180,E1 -1519.836,E2 -1519.836} C_VEL
LIN {X 0,Y 587.366,Z 286.598,A -85,B 0,C 180,E1 -1520.617,E2 -1520.617} C_VEL
LIN {X 0,Y 587.322,Z 295.111,A -85,B 0,C 180,E1 -1521.397,E2 -1521.397} C_VEL
LIN {X 0,Y 587.274,Z 302.959,A -85,B 0,C 180,E1 -1522.263,E2 -1522.263} C_VEL
LIN {X 0,Y 587.23,Z 309.468,A -85,B 0,C 180,E1 -1523.126,E2 -1523.126} C_VEL
LIN {X 0,Y 587.237,Z 315.866,A -85,B 0,C 180,E1 -1524.161,E2 -1524.161} C_VEL
LIN {X 0,Y 587.147,Z 320.949,A -85,B 0,C 180,E1 -1525.194,E2 -1525.194} C_VEL
LIN {X 0,Y 587.213,Z 324.895,A -85,B 0,C 180,E1 -1526.226,E2 -1526.226} C_VEL
LIN {X 0,Y 587.132,Z 327.808,A -85,B 0,C 180,E1 -1527.256,E2 -1527.256} C_VEL
LIN {X 0,Y 587.141,Z 329.199,A -85,B 0,C 180,E1 -1527.942,E2 -1527.942} C_VEL
LIN {X 0,Y 587.14,Z 330.785,A -85,B 0,C 180,E1 -1529.314,E2 -1529.314} C_VEL
LIN {X 0,Y 587.137,Z 331,A -85,B 0,C 180,E1 -1530,E2 -1530} C_VEL
LIN {X 0,Y 587.147,Z 330.186,A -85,B 0,C 180,E1 -1531.372,E2 -1531.372} C_VEL
LIN {X 0,Y 587.141,Z 329.2,A -85,B 0,C 180,E1 -1532.058,E2 -1532.058} C_VEL
LIN {X 0,Y 587.132,Z 327.81,A -85,B 0,C 180,E1 -1532.744,E2 -1532.744} C_VEL
LIN {X 0,Y 587.213,Z 324.896,A -85,B 0,C 180,E1 -1533.774,E2 -1533.774} C_VEL
LIN {X 0,Y 587.147,Z 320.949,A -85,B 0,C 180,E1 -1534.806,E2 -1534.806} C_VEL
LIN {X 0,Y 587.218,Z 314.877,A -85,B 0,C 180,E1 -1536.011,E2 -1536.011} C_VEL
LIN {X 0,Y 587.245,Z 308.237,A -85,B 0,C 180,E1 -1537.046,E2 -1537.046} C_VEL
LIN {X 0,Y 587.299,Z 299.99,A -85,B 0,C 180,E1 -1538.083,E2 -1538.083} C_VEL
LIN {X 0,Y 587.343,Z 291.538,A -85,B 0,C 180,E1 -1538.949,E2 -1538.949} C_VEL
LIN {X 0,Y 587.413,Z 281.097,A -85,B 0,C 180,E1 -1539.816,E2 -1539.816} C_VEL
LIN {X 0,Y 587.48,Z 270.755,A -85,B 0,C 180,E1 -1540.512,E2 -1540.512} C_VEL
LIN {X 0,Y 587.561,Z 258.815,A -85,B 0,C 180,E1 -1541.149,E2 -1541.149} C_VEL
LIN {X 0,Y 587.63,Z 246.596,A -85,B 0,C 180,E1 -1541.639,E2 -1541.639} C_VEL
LIN {X 0,Y 587.702,Z 233.432,A -85,B 0,C 180,E1 -1542.014,E2 -1542.014} C_VEL
LIN {X 0,Y 587.773,Z 221.081,A -85,B 0,C 180,E1 -1542.232,E2 -1542.232} C_VEL
LIN {X 0,Y 587.726,Z 120.479,A -85,B 0,C 180,E1 -1543.468,E2 -1543.468} C_VEL
LIN {X 0,Y 587.408,Z 118.269,A -85,B 0,C 180,E1 -1543.514,E2 -1543.514} C_VEL
LIN {X 0,Y 587.547,Z 96.603,A -85,B 0,C 180,E1 -1546.326,E2 -1546.326} C_VEL
LIN {X 0,Y 587.663,Z 77.497,A -85,B 0,C 180,E1 -1548.838,E2 -1548.838} C_VEL
LIN {X 0,Y 587.794,Z 58.137,A -85,B 0,C 180,E1 -1551.394,E2 -1551.394} C_VEL
LIN {X 0,Y 587.862,Z 42.789,A -85,B 0,C 180,E1 -1553.423,E2 -1553.423} C_VEL
LIN {X 0,Y 587.348,Z 39.323,A -85,B 0,C 180,E1 -1553.912,E2 -1553.912} C_VEL
LIN {X 0,Y 587.339,Z 39.327,A -85,B 0,C 180,E1 -1556.279,E2 -1556.279} C_VEL
LIN {X 0,Y 587.352,Z 39.317,A -85,B 0,C 180,E1 -1559.133,E2 -1559.133} C_VEL
LIN {X 0,Y 587.345,Z 39.322,A -85,B 0,C 180,E1 -1561.835,E2 -1561.835} C_VEL
LIN {X 0,Y 587.348,Z 39.323,A -85,B 0,C 180,E1 -1564.347,E2 -1564.347} C_VEL
LIN {X 0,Y 587.346,Z 39.322,A -85,B 0,C 180,E1 -1567.608,E2 -1567.608} C_VEL
LIN {X 0,Y 587.314,Z 39.325,A -85,B 0,C 180,E1 -1570.255,E2 -1570.255} C_VEL
LIN {X 0,Y 587.316,Z 39.322,A -85,B 0,C 180,E1 -1573.118,E2 -1573.118} C_VEL
LIN {X 0,Y 587.316,Z 39.324,A -85,B 0,C 180,E1 -1576.049,E2 -1576.049} C_VEL
LIN {X 0,Y 587.337,Z 39.32,A -85,B 0,C 180,E1 -1578.925,E2 -1578.925} C_VEL
LIN {X 0,Y 587.331,Z 39.327,A -85,B 0,C 180,E1 -1581.52,E2 -1581.52} C_VEL
LIN {X 0,Y 587.296,Z 39.324,A -85,B 0,C 180,E1 -1584.1,E2 -1584.1} C_VEL
LIN {X 0,Y 587.34,Z 39.323,A -85,B 0,C 180,E1 -1586.889,E2 -1586.889} C_VEL
LIN {X 0,Y 587.337,Z 39.318,A -85,B 0,C 180,E1 -1589.83,E2 -1589.83} C_VEL
LIN {X 0,Y 587.356,Z 39.317,A -85,B 0,C 180,E1 -1592.307,E2 -1592.307} C_VEL
LIN {X 0,Y 587.355,Z 39.32,A -85,B 0,C 180,E1 -1595.241,E2 -1595.241} C_VEL
LIN {X 0,Y 587.326,Z 39.322,A -85,B 0,C 180,E1 -1598.226,E2 -1598.226} C_VEL
LIN {X 0,Y 587.35,Z 39.319,A -85,B 0,C 180,E1 -1601.151,E2 -1601.151} C_VEL
LIN {X 0,Y 587.325,Z 39.322,A -85,B 0,C 180,E1 -1604.025,E2 -1604.025} C_VEL
LIN {X 0,Y 587.36,Z 39.322,A -85,B 0,C 180,E1 -1606.154,E2 -1606.154} C_VEL
LIN {X 0,Y 587.345,Z 39.318,A -85,B 0,C 180,E1 -1608.962,E2 -1608.962} C_VEL
LIN {X 0,Y 587.369,Z 39.318,A -85,B 0,C 180,E1 -1611.745,E2 -1611.745} C_VEL
LIN {X 0,Y 587.355,Z 39.319,A -85,B 0,C 180,E1 -1614.507,E2 -1614.507} C_VEL
LIN {X 0,Y 587.374,Z 39.315,A -85,B 0,C 180,E1 -1617.257,E2 -1617.257} C_VEL
LIN {X 0,Y 587.384,Z 39.32,A -85,B 0,C 180,E1 -1620,E2 -1620} C_VEL
LIN {X 0,Y 587.371,Z 39.314,A -85,B 0,C 180,E1 -1622.743,E2 -1622.743} C_VEL
LIN {X 0,Y 587.355,Z 39.324,A -85,B 0,C 180,E1 -1625.493,E2 -1625.493} C_VEL
LIN {X 0,Y 587.343,Z 39.317,A -85,B 0,C 180,E1 -1628.256,E2 -1628.256} C_VEL
LIN {X 0,Y 587.354,Z 39.322,A -85,B 0,C 180,E1 -1631.133,E2 -1631.133} C_VEL
LIN {X 0,Y 587.361,Z 39.315,A -85,B 0,C 180,E1 -1634.257,E2 -1634.257} C_VEL
LIN {X 0,Y 587.349,Z 39.322,A -85,B 0,C 180,E1 -1637.406,E2 -1637.406} C_VEL
LIN {X 0,Y 587.304,Z 39.323,A -85,B 0,C 180,E1 -1638.3,E2 -1638.3} C_VEL
LIN {X 0,Y 586.667,Z 39.409,A -85,B 0,C 180,E1 -1638.872,E2 -1638.872} C_VEL
LIN {X 0,Y 583.848,Z 39.763,A -85,B 0,C 180,E1 -1639.801,E2 -1639.801} C_VEL
LIN {X 0,Y 581.439,Z 40.063,A -85,B 0,C 180,E1 -1640.548,E2 -1640.548} C_VEL
LIN {X 0,Y 580.383,Z 40.192,A -85,B 0,C 180,E1 -1641.124,E2 -1641.124} C_VEL
LIN {X 0,Y 580.287,Z 40.201,A -85,B 0,C 180,E1 -1641.32,E2 -1641.32} C_VEL
LIN {X 0,Y 580.3,Z 40.197,A -85,B 0,C 180,E1 -1644.316,E2 -1644.316} C_VEL
LIN {X 0,Y 580.27,Z 40.207,A -85,B 0,C 180,E1 -1646.624,E2 -1646.624} C_VEL
LIN {X 0,Y 580.3,Z 40.196,A -85,B 0,C 180,E1 -1649.309,E2 -1649.309} C_VEL
LIN {X 0,Y 580.3,Z 40.2,A -85,B 0,C 180,E1 -1652.2,E2 -1652.2} C_VEL
LIN {X 0,Y 580.282,Z 40.203,A -85,B 0,C 180,E1 -1654.697,E2 -1654.697} C_VEL
LIN {X 0,Y 580.289,Z 40.196,A -85,B 0,C 180,E1 -1657.269,E2 -1657.269} C_VEL
LIN {X 0,Y 580.29,Z 40.203,A -85,B 0,C 180,E1 -1660.27,E2 -1660.27} C_VEL
LIN {X 0,Y 580.268,Z 40.201,A -85,B 0,C 180,E1 -1663.389,E2 -1663.389} C_VEL
LIN {X 0,Y 580.243,Z 40.206,A -85,B 0,C 180,E1 -1666.338,E2 -1666.338} C_VEL
LIN {X 0,Y 580.294,Z 40.197,A -85,B 0,C 180,E1 -1669.156,E2 -1669.156} C_VEL
LIN {X 0,Y 580.282,Z 40.204,A -85,B 0,C 180,E1 -1671.928,E2 -1671.928} C_VEL
LIN {X 0,Y 580.25,Z 40.202,A -85,B 0,C 180,E1 -1674.452,E2 -1674.452} C_VEL
LIN {X 0,Y 580.288,Z 40.2,A -85,B 0,C 180,E1 -1676.975,E2 -1676.975} C_VEL
LIN {X 0,Y 580.282,Z 40.208,A -85,B 0,C 180,E1 -1679.424,E2 -1679.424} C_VEL
LIN {X 0,Y 580.314,Z 40.275,A -85,B 0,C 180,E1 -1682.453,E2 -1682.453} C_VEL
LIN {X 0,Y 580.329,Z 53.075,A -85,B 0,C 180,E1 -1684.921,E2 -1684.921} C_VEL
LIN {X 0,Y 580.278,Z 60.84,A -85,B 0,C 180,E1 -1686.394,E2 -1686.394} C_VEL
LIN {X 0,Y 580.953,Z 66.043,A -85,B 0,C 180,E1 -1686.486,E2 -1686.486} C_VEL
LIN {X 0,Y 580.779,Z 167.172,A -85,B 0,C 180,E1 -1687.757,E2 -1687.757} C_VEL
LIN {X 0,Y 580.735,Z 180.921,A -85,B 0,C 180,E1 -1688.083,E2 -1688.083} C_VEL
LIN {X 0,Y 580.66,Z 193.422,A -85,B 0,C 180,E1 -1688.523,E2 -1688.523} C_VEL
LIN {X 0,Y 580.535,Z 205.293,A -85,B 0,C 180,E1 -1689.09,E2 -1689.09} C_VEL
LIN {X 0,Y 580.41,Z 217.012,A -85,B 0,C 180,E1 -1689.812,E2 -1689.812} C_VEL
LIN {X 0,Y 580.363,Z 227.044,A -85,B 0,C 180,E1 -1690.585,E2 -1690.585} C_VEL
LIN {X 0,Y 580.298,Z 236.322,A -85,B 0,C 180,E1 -1691.463,E2 -1691.463} C_VEL
LIN {X 0,Y 580.198,Z 245.623,A -85,B 0,C 180,E1 -1692.554,E2 -1692.554} C_VEL
LIN {X 0,Y 580.107,Z 253.065,A -85,B 0,C 180,E1 -1693.647,E2 -1693.647} C_VEL
LIN {X 0,Y 580.107,Z 257.985,A -85,B 0,C 180,E1 -1694.542,E2 -1694.542} C_VEL
LIN {X 0,Y 580.087,Z 263.229,A -85,B 0,C 180,E1 -1695.751,E2 -1695.751} C_VEL
LIN {X 0,Y 580.077,Z 266.322,A -85,B 0,C 180,E1 -1696.691,E2 -1696.691} C_VEL
LIN {X 0,Y 580.056,Z 268.102,A -85,B 0,C 180,E1 -1697.403,E2 -1697.403} C_VEL
LIN {X 0,Y 580.054,Z 269.444,A -85,B 0,C 180,E1 -1698.113,E2 -1698.113} C_VEL
LIN {X 0,Y 580.071,Z 270.485,A -85,B 0,C 180,E1 -1698.925,E2 -1698.925} C_VEL
LIN {X 0,Y 580.057,Z 270.964,A -85,B 0,C 180,E1 -1700.234,E2 -1700.234} C_VEL
LIN {X 0,Y 580.059,Z 269.947,A -85,B 0,C 180,E1 -1701.64,E2 -1701.64} C_VEL
LIN {X 0,Y 580.065,Z 268.817,A -85,B 0,C 180,E1 -1702.341,E2 -1702.341} C_VEL
LIN {X 0,Y 580.107,Z 266.229,A -85,B 0,C 180,E1 -1703.429,E2 -1703.429} C_VEL
LIN {X 0,Y 580.111,Z 262.869,A -85,B 0,C 180,E1 -1704.438,E2 -1704.438} C_VEL
LIN {X 0,Y 580.118,Z 258.314,A -85,B 0,C 180,E1 -1705.484,E2 -1705.484} C_VEL
LIN {X 0,Y 580.129,Z 251.435,A -85,B 0,C 180,E1 -1706.701,E2 -1706.701} C_VEL
LIN {X 0,Y 580.197,Z 244.011,A -85,B 0,C 180,E1 -1707.744,E2 -1707.744} C_VEL
LIN {X 0,Y 580.269,Z 236.464,A -85,B 0,C 180,E1 -1708.612,E2 -1708.612} C_VEL
LIN {X 0,Y 580.335,Z 227.355,A -85,B 0,C 180,E1 -1709.48,E2 -1709.48} C_VEL
LIN {X 0,Y 580.397,Z 217.27,A -85,B 0,C 180,E1 -1710.26,E2 -1710.26} C_VEL
LIN {X 0,Y 580.544,Z 206.11,A -85,B 0,C 180,E1 -1710.954,E2 -1710.954} C_VEL
LIN {X 0,Y 580.631,Z 193.603,A -85,B 0,C 180,E1 -1711.561,E2 -1711.561} C_VEL
LIN {X 0,Y 580.671,Z 180.685,A -85,B 0,C 180,E1 -1712.016,E2 -1712.016} C_VEL
LIN {X 0,Y 580.783,Z 167.889,A -85,B 0,C 180,E1 -1712.319,E2 -1712.319} C_VEL
LIN {X 0,Y 580.914,Z 106.649,A -85,B 0,C 180,E1 -1713.099,E2 -1713.099} C_VEL
LIN {X 0,Y 580.784,Z 64.115,A -85,B 0,C 180,E1 -1713.632,E2 -1713.632} C_VEL
LIN {X 0,Y 580.263,Z 60.875,A -85,B 0,C 180,E1 -1713.689,E2 -1713.689} C_VEL
LIN {X 0,Y 580.375,Z 47.373,A -85,B 0,C 180,E1 -1716.257,E2 -1716.257} C_VEL
LIN {X 0,Y 580.317,Z 40.197,A -85,B 0,C 180,E1 -1717.656,E2 -1717.656} C_VEL
LIN {X 0,Y 580.302,Z 40.202,A -85,B 0,C 180,E1 -1720.467,E2 -1720.467} C_VEL
LIN {X 0,Y 580.306,Z 40.203,A -85,B 0,C 180,E1 -1722.591,E2 -1722.591} C_VEL
LIN {X 0,Y 580.289,Z 40.203,A -85,B 0,C 180,E1 -1724.734,E2 -1724.734} C_VEL
LIN {X 0,Y 580.295,Z 40.196,A -85,B 0,C 180,E1 -1727.625,E2 -1727.625} C_VEL
LIN {X 0,Y 580.29,Z 40.198,A -85,B 0,C 180,E1 -1729.823,E2 -1729.823} C_VEL
LIN {X 0,Y 580.275,Z 40.204,A -85,B 0,C 180,E1 -1732.053,E2 -1732.053} C_VEL
LIN {X 0,Y 580.307,Z 40.194,A -85,B 0,C 180,E1 -1735.08,E2 -1735.08} C_VEL
LIN {X 0,Y 580.303,Z 40.203,A -85,B 0,C 180,E1 -1738.186,E2 -1738.186} C_VEL
LIN {X 0,Y 580.287,Z 40.197,A -85,B 0,C 180,E1 -1740.695,E2 -1740.695} C_VEL
LIN {X 0,Y 580.305,Z 40.196,A -85,B 0,C 180,E1 -1743.316,E2 -1743.316} C_VEL
LIN {X 0,Y 580.263,Z 40.209,A -85,B 0,C 180,E1 -1745.758,E2 -1745.758} C_VEL
LIN {X 0,Y 580.29,Z 40.199,A -85,B 0,C 180,E1 -1748.147,E2 -1748.147} C_VEL
LIN {X 0,Y 580.3,Z 40.195,A -85,B 0,C 180,E1 -1750.844,E2 -1750.844} C_VEL
LIN {X 0,Y 580.275,Z 40.206,A -85,B 0,C 180,E1 -1753.659,E2 -1753.659} C_VEL
LIN {X 0,Y 580.277,Z 40.198,A -85,B 0,C 180,E1 -1756.61,E2 -1756.61} C_VEL
LIN {X 0,Y 580.3,Z 40.202,A -85,B 0,C 180,E1 -1759.157,E2 -1759.157} C_VEL
LIN {X 0,Y 580.292,Z 40.197,A -85,B 0,C 180,E1 -1761.927,E2 -1761.927} C_VEL
LIN {X 0,Y 580.257,Z 40.201,A -85,B 0,C 180,E1 -1764.453,E2 -1764.453} C_VEL
LIN {X 0,Y 580.292,Z 40.205,A -85,B 0,C 180,E1 -1766.975,E2 -1766.975} C_VEL
LIN {X 0,Y 580.3,Z 40.198,A -85,B 0,C 180,E1 -1769.425,E2 -1769.425} C_VEL
LIN {X 0,Y 580.301,Z 40.196,A -85,B 0,C 180,E1 -1772.142,E2 -1772.142} C_VEL
LIN {X 0,Y 580.326,Z 40.194,A -85,B 0,C 180,E1 -1775.27,E2 -1775.27} C_VEL
LIN {X 0,Y 580.276,Z 40.199,A -85,B 0,C 180,E1 -1777.948,E2 -1777.948} C_VEL
LIN {X 0,Y 580.302,Z 40.199,A -85,B 0,C 180,E1 -1780.914,E2 -1780.914} C_VEL
LIN {X 0,Y 580.274,Z 40.2,A -85,B 0,C 180,E1 -1783.825,E2 -1783.825} C_VEL
LIN {X 0,Y 580.33,Z 40.195,A -85,B 0,C 180,E1 -1785.983,E2 -1785.983} C_VEL
LIN {X 0,Y 580.312,Z 40.195,A -85,B 0,C 180,E1 -1788.827,E2 -1788.827} C_VEL
LIN {X 0,Y 580.317,Z 40.195,A -85,B 0,C 180,E1 -1791.644,E2 -1791.644} C_VEL
LIN {X 0,Y 580.288,Z 40.201,A -85,B 0,C 180,E1 -1793.742,E2 -1793.742} C_VEL
LIN {X 0,Y 580.272,Z 40.205,A -85,B 0,C 180,E1 -1795.833,E2 -1795.833} C_VEL
LIN {X 0,Y 580.341,Z 40.2,A -85,B 0,C 180,E1 -1797.918,E2 -1797.918} C_VEL
LIN {X 0,Y 580.361,Z 40.187,A -85,B 0,C 180,E1 -1800.694,E2 -1800.694} C_VEL
LIN {X 0,Y 580.283,Z 40.203,A -85,B 0,C 180,E1 -1803.472,E2 -1803.472} C_VEL
LIN {X 0,Y 580.321,Z 40.201,A -85,B 0,C 180,E1 -1805.56,E2 -1805.56} C_VEL
LIN {X 0,Y 580.315,Z 40.193,A -85,B 0,C 180,E1 -1808.356,E2 -1808.356} C_VEL
LIN {X 0,Y 580.307,Z 40.2,A -85,B 0,C 180,E1 -1811.191,E2 -1811.191} C_VEL
LIN {X 0,Y 580.322,Z 40.193,A -85,B 0,C 180,E1 -1814.017,E2 -1814.017} C_VEL
LIN {X 0,Y 580.319,Z 40.197,A -85,B 0,C 180,E1 -1816.914,E2 -1816.914} C_VEL
LIN {X 0,Y 580.291,Z 40.197,A -85,B 0,C 180,E1 -1819.823,E2 -1819.823} C_VEL
LIN {X 0,Y 580.275,Z 40.198,A -85,B 0,C 180,E1 -1822.053,E2 -1822.053} C_VEL
LIN {X 0,Y 580.306,Z 40.202,A -85,B 0,C 180,E1 -1825.08,E2 -1825.08} C_VEL
LIN {X 0,Y 580.287,Z 40.198,A -85,B 0,C 180,E1 -1828.186,E2 -1828.186} C_VEL
LIN {X 0,Y 580.288,Z 40.206,A -85,B 0,C 180,E1 -1830.694,E2 -1830.694} C_VEL
LIN {X 0,Y 580.288,Z 40.198,A -85,B 0,C 180,E1 -1833.313,E2 -1833.313} C_VEL
LIN {X 0,Y 580.249,Z 40.202,A -85,B 0,C 180,E1 -1835.756,E2 -1835.756} C_VEL
LIN {X 0,Y 580.289,Z 40.201,A -85,B 0,C 180,E1 -1838.146,E2 -1838.146} C_VEL
LIN {X 0,Y 580.299,Z 40.198,A -85,B 0,C 180,E1 -1840.844,E2 -1840.844} C_VEL
LIN {X 0,Y 580.277,Z 40.199,A -85,B 0,C 180,E1 -1843.658,E2 -1843.658} C_VEL
LIN {X 0,Y 580.248,Z 40.205,A -85,B 0,C 180,E1 -1846.613,E2 -1846.613} C_VEL
LIN {X 0,Y 580.299,Z 40.195,A -85,B 0,C 180,E1 -1849.156,E2 -1849.156} C_VEL
LIN {X 0,Y 580.291,Z 40.205,A -85,B 0,C 180,E1 -1851.927,E2 -1851.927} C_VEL
LIN {X 0,Y 580.255,Z 40.202,A -85,B 0,C 180,E1 -1854.453,E2 -1854.453} C_VEL
LIN {X 0,Y 580.292,Z 40.196,A -85,B 0,C 180,E1 -1856.975,E2 -1856.975} C_VEL
LIN {X 0,Y 580.29,Z 40.201,A -85,B 0,C 180,E1 -1859.424,E2 -1859.424} C_VEL
LIN {X 0,Y 580.296,Z 40.198,A -85,B 0,C 180,E1 -1862.142,E2 -1862.142} C_VEL
LIN {X 0,Y 580.323,Z 40.2,A -85,B 0,C 180,E1 -1865.27,E2 -1865.27} C_VEL
LIN {X 0,Y 580.333,Z 40.364,A -85,B 0,C 180,E1 -1865.97,E2 -1865.97} C_VEL
LIN {X 0,Y 580.921,Z 43.878,A -85,B 0,C 180,E1 -1866.469,E2 -1866.469} C_VEL
LIN {X 0,Y 580.78,Z 63.447,A -85,B 0,C 180,E1 -1869.085,E2 -1869.085} C_VEL
LIN {X 0,Y 580.705,Z 82.948,A -85,B 0,C 180,E1 -1871.659,E2 -1871.659} C_VEL
LIN {X 0,Y 580.51,Z 104.791,A -85,B 0,C 180,E1 -1874.553,E2 -1874.553} C_VEL
LIN {X 0,Y 580.422,Z 118.353,A -85,B 0,C 180,E1 -1876.331,E2 -1876.331} C_VEL
LIN {X 0,Y 580.95,Z 124.494,A -85,B 0,C 180,E1 -1876.422,E2 -1876.422} C_VEL
LIN {X 0,Y 580.785,Z 226.938,A -85,B 0,C 180,E1 -1877.708,E2 -1877.708} C_VEL
LIN {X 0,Y 580.741,Z 240.213,A -85,B 0,C 180,E1 -1878.017,E2 -1878.017} C_VEL
LIN {X 0,Y 580.656,Z 252.372,A -85,B 0,C 180,E1 -1878.436,E2 -1878.436} C_VEL
LIN {X 0,Y 580.58,Z 264.624,A -85,B 0,C 180,E1 -1879.009,E2 -1879.009} C_VEL
LIN {X 0,Y 580.436,Z 276.197,A -85,B 0,C 180,E1 -1879.712,E2 -1879.712} C_VEL
LIN {X 0,Y 580.346,Z 286.6,A -85,B 0,C 180,E1 -1880.503,E2 -1880.503} C_VEL
LIN {X 0,Y 580.271,Z 295.111,A -85,B 0,C 180,E1 -1881.292,E2 -1881.292} C_VEL
LIN {X 0,Y 580.222,Z 302.96,A -85,B 0,C 180,E1 -1882.168,E2 -1882.168} C_VEL
LIN {X 0,Y 580.154,Z 310.651,A -85,B 0,C 180,E1 -1883.222,E2 -1883.222} C_VEL
LIN {X 0,Y 580.139,Z 317.679,A -85,B 0,C 180,E1 -1884.438,E2 -1884.438} C_VEL
LIN {X 0,Y 580.108,Z 322.372,A -85,B 0,C 180,E1 -1885.483,E2 -1885.483} C_VEL
LIN {X 0,Y 580.123,Z 325.957,A -85,B 0,C 180,E1 -1886.527,E2 -1886.527} C_VEL
LIN {X 0,Y 580.043,Z 327.808,A -85,B 0,C 180,E1 -1887.222,E2 -1887.222} C_VEL
LIN {X 0,Y 580.04,Z 329.197,A -85,B 0,C 180,E1 -1887.917,E2 -1887.917} C_VEL
LIN {X 0,Y 580.04,Z 330.785,A -85,B 0,C 180,E1 -1889.306,E2 -1889.306} C_VEL
LIN {X 0,Y 580.037,Z 331,A -85,B 0,C 180,E1 -1890,E2 -1890} C_VEL
LIN {X 0,Y 580.047,Z 330.186,A -85,B 0,C 180,E1 -1891.389,E2 -1891.389} C_VEL
LIN {X 0,Y 580.04,Z 329.199,A -85,B 0,C 180,E1 -1892.083,E2 -1892.083} C_VEL
LIN {X 0,Y 580.043,Z 327.81,A -85,B 0,C 180,E1 -1892.778,E2 -1892.778} C_VEL
LIN {X 0,Y 580.11,Z 324.896,A -85,B 0,C 180,E1 -1893.821,E2 -1893.821} C_VEL
LIN {X 0,Y 580.053,Z 320.949,A -85,B 0,C 180,E1 -1894.865,E2 -1894.865} C_VEL
LIN {X 0,Y 580.139,Z 314.877,A -85,B 0,C 180,E1 -1896.085,E2 -1896.085} C_VEL
LIN {X 0,Y 580.184,Z 308.237,A -85,B 0,C 180,E1 -1897.132,E2 -1897.132} C_VEL
LIN {X 0,Y 580.25,Z 299.991,A -85,B 0,C 180,E1 -1898.182,E2 -1898.182} C_VEL
LIN {X 0,Y 580.308,Z 291.539,A -85,B 0,C 180,E1 -1899.058,E2 -1899.058} C_VEL
LIN {X 0,Y 580.416,Z 281.097,A -85,B 0,C 180,E1 -1899.936,E2 -1899.936} C_VEL
LIN {X 0,Y 580.501,Z 270.753,A -85,B 0,C 180,E1 -1900.64,E2 -1900.64} C_VEL
LIN {X 0,Y 580.596,Z 259.243,A -85,B 0,C 180,E1 -1901.264,E2 -1901.264} C_VEL
LIN {X 0,Y 580.682,Z 246.47,A -85,B 0,C 180,E1 -1901.785,E2 -1901.785} C_VEL
LIN {X 0,Y 580.776,Z 233.43,A -85,B 0,C 180,E1 -1902.16,E2 -1902.16} C_VEL
LIN {X 0,Y 580.857,Z 221.081,A -85,B 0,C 180,E1 -1902.38,E2 -1902.38} C_VEL
LIN {X 0,Y 580.819,Z 121.151,A -85,B 0,C 180,E1 -1903.623,E2 -1903.623} C_VEL
LIN {X 0,Y 580.429,Z 118.269,A -85,B 0,C 180,E1 -1903.68,E2 -1903.68} C_VEL
LIN {X 0,Y 580.6,Z 95.239,A -85,B 0,C 180,E1 -1906.708,E2 -1906.708} C_VEL
LIN {X 0,Y 580.698,Z 77.371,A -85,B 0,C 180,E1 -1909.073,E2 -1909.073} C_VEL
LIN {X 0,Y 580.82,Z 57.798,A -85,B 0,C 180,E1 -1911.657,E2 -1911.657} C_VEL
LIN {X 0,Y 580.896,Z 43.829,A -85,B 0,C 180,E1 -1913.532,E2 -1913.532} C_VEL
LIN {X 0,Y 580.313,Z 40.202,A -85,B 0,C 180,E1 -1914.078,E2 -1914.078} C_VEL
LIN {X 0,Y 580.279,Z 40.205,A -85,B 0,C 180,E1 -1916.623,E2 -1916.623} C_VEL
LIN {X 0,Y 580.303,Z 40.195,A -85,B 0,C 180,E1 -1919.309,E2 -1919.309} C_VEL
LIN {X 0,Y 580.3,Z 40.205,A -85,B 0,C 180,E1 -1922.201,E2 -1922.201} C_VEL
LIN {X 0,Y 580.292,Z 40.198,A -85,B 0,C 180,E1 -1924.696,E2 -1924.696} C_VEL
LIN {X 0,Y 580.301,Z 40.196,A -85,B 0,C 180,E1 -1927.269,E2 -1927.269} C_VEL
LIN {X 0,Y 580.294,Z 40.199,A -85,B 0,C 180,E1 -1930.27,E2 -1930.27} C_VEL
LIN {X 0,Y 580.28,Z 40.197,A -85,B 0,C 180,E1 -1932.706,E2 -1932.706} C_VEL
LIN {X 0,Y 580.259,Z 40.209,A -85,B 0,C 180,E1 -1935.611,E2 -1935.611} C_VEL
LIN {X 0,Y 580.283,Z 40.198,A -85,B 0,C 180,E1 -1938.231,E2 -1938.231} C_VEL
LIN {X 0,Y 580.281,Z 40.2,A -85,B 0,C 180,E1 -1940.965,E2 -1940.965} C_VEL
LIN {X 0,Y 580.272,Z 40.203,A -85,B 0,C 180,E1 -1943.596,E2 -1943.596} C_VEL
LIN {X 0,Y 580.305,Z 40.194,A -85,B 0,C 180,E1 -1946.144,E2 -1946.144} C_VEL
LIN {X 0,Y 580.279,Z 40.2,A -85,B 0,C 180,E1 -1948.615,E2 -1948.615} C_VEL
LIN {X 0,Y 580.296,Z 40.205,A -85,B 0,C 180,E1 -1951.024,E2 -1951.024} C_VEL
LIN {X 0,Y 580.294,Z 40.196,A -85,B 0,C 180,E1 -1953.666,E2 -1953.666} C_VEL
LIN {X 0,Y 580.302,Z 40.195,A -85,B 0,C 180,E1 -1955.684,E2 -1955.684} C_VEL
LIN {X 0,Y 580.29,Z 40.205,A -85,B 0,C 180,E1 -1958.695,E2 -1958.695} C_VEL
LIN {X 0,Y 580.302,Z 40.199,A -85,B 0,C 180,E1 -1960.913,E2 -1960.913} C_VEL
LIN {X 0,Y 580.28,Z 40.198,A -85,B 0,C 180,E1 -1963.825,E2 -1963.825} C_VEL
LIN {X 0,Y 580.328,Z 40.195,A -85,B 0,C 180,E1 -1965.983,E2 -1965.983} C_VEL
LIN {X 0,Y 580.311,Z 40.196,A -85,B 0,C 180,E1 -1968.827,E2 -1968.827} C_VEL
LIN {X 0,Y 580.332,Z 40.193,A -85,B 0,C 180,E1 -1971.644,E2 -1971.644} C_VEL
LIN {X 0,Y 580.322,Z 40.196,A -85,B 0,C 180,E1 -1974.44,E2 -1974.44} C_VEL
LIN {X 0,Y 580.34,Z 40.199,A -85,B 0,C 180,E1 -1977.918,E2 -1977.918} C_VEL
LIN {X 0,Y 580.361,Z 40.188,A -85,B 0,C 180,E1 -1980.694,E2 -1980.694} C_VEL
LIN {X 0,Y 580.282,Z 40.203,A -85,B 0,C 180,E1 -1983.472,E2 -1983.472} C_VEL
LIN {X 0,Y 580.32,Z 40.201,A -85,B 0,C 180,E1 -1985.56,E2 -1985.56} C_VEL
LIN {X 0,Y 580.313,Z 40.193,A -85,B 0,C 180,E1 -1988.356,E2 -1988.356} C_VEL
LIN {X 0,Y 580.306,Z 40.201,A -85,B 0,C 180,E1 -1991.191,E2 -1991.191} C_VEL
LIN {X 0,Y 580.321,Z 40.192,A -85,B 0,C 180,E1 -1994.017,E2 -1994.017} C_VEL
LIN {X 0,Y 580.318,Z 40.199,A -85,B 0,C 180,E1 -1996.914,E2 -1996.914} C_VEL
LIN {X 0,Y 580.289,Z 40.197,A -85,B 0,C 180,E1 -1999.823,E2 -1999.823} C_VEL
LIN {X 0,Y 580.287,Z 40.201,A -85,B 0,C 180,E1 -2001.32,E2 -2001.32} C_VEL
LIN {X 0,Y 579.587,Z 40.286,A -85,B 0,C 180,E1 -2001.899,E2 -2001.899} C_VEL
LIN {X 0,Y 576.707,Z 40.651,A -85,B 0,C 180,E1 -2002.838,E2 -2002.838} C_VEL
LIN {X 0,Y 574.313,Z 40.944,A -85,B 0,C 180,E1 -2003.595,E2 -2003.595} C_VEL
LIN {X 0,Y 573.315,Z 41.066,A -85,B 0,C 180,E1 -2004.179,E2 -2004.179} C_VEL
LIN {X 0,Y 573.249,Z 41.076,A -85,B 0,C 180,E1 -2004.376,E2 -2004.376} C_VEL
LIN {X 0,Y 573.206,Z 41.084,A -85,B 0,C 180,E1 -2006.978,E2 -2006.978} C_VEL
LIN {X 0,Y 573.246,Z 41.074,A -85,B 0,C 180,E1 -2009.487,E2 -2009.487} C_VEL
LIN {X 0,Y 573.255,Z 41.08,A -85,B 0,C 180,E1 -2012.645,E2 -2012.645} C_VEL
LIN {X 0,Y 573.196,Z 41.081,A -85,B 0,C 180,E1 -2015.189,E2 -2015.189} C_VEL
LIN {X 0,Y 573.232,Z 41.078,A -85,B 0,C 180,E1 -2017.808,E2 -2017.808} C_VEL
LIN {X 0,Y 573.247,Z 41.076,A -85,B 0,C 180,E1 -2020.525,E2 -2020.525} C_VEL
LIN {X 0,Y 573.231,Z 41.077,A -85,B 0,C 180,E1 -2023.36,E2 -2023.36} C_VEL
LIN {X 0,Y 573.212,Z 41.082,A -85,B 0,C 180,E1 -2026.335,E2 -2026.335} C_VEL
LIN {X 0,Y 573.227,Z 41.077,A -85,B 0,C 180,E1 -2028.542,E2 -2028.542} C_VEL
LIN {X 0,Y 573.234,Z 41.079,A -85,B 0,C 180,E1 -2031.297,E2 -2031.297} C_VEL
LIN {X 0,Y 573.194,Z 41.085,A -85,B 0,C 180,E1 -2034.021,E2 -2034.021} C_VEL
LIN {X 0,Y 573.23,Z 41.077,A -85,B 0,C 180,E1 -2036.515,E2 -2036.515} C_VEL
LIN {X 0,Y 573.221,Z 41.084,A -85,B 0,C 180,E1 -2039.119,E2 -2039.119} C_VEL
LIN {X 0,Y 573.25,Z 41.079,A -85,B 0,C 180,E1 -2041.972,E2 -2041.972} C_VEL
LIN {X 0,Y 573.283,Z 41.214,A -85,B 0,C 180,E1 -2042.383,E2 -2042.383} C_VEL
LIN {X 0,Y 573.323,Z 52.517,A -85,B 0,C 180,E1 -2044.593,E2 -2044.593} C_VEL
LIN {X 0,Y 573.239,Z 60.888,A -85,B 0,C 180,E1 -2046.233,E2 -2046.233} C_VEL
LIN {X 0,Y 574.076,Z 66.612,A -85,B 0,C 180,E1 -2046.328,E2 -2046.328} C_VEL
LIN {X 0,Y 573.835,Z 167.659,A -85,B 0,C 180,E1 -2047.616,E2 -2047.616} C_VEL
LIN {X 0,Y 573.79,Z 181.248,A -85,B 0,C 180,E1 -2047.945,E2 -2047.945} C_VEL
LIN {X 0,Y 573.684,Z 193.645,A -85,B 0,C 180,E1 -2048.39,E2 -2048.39} C_VEL
LIN {X 0,Y 573.548,Z 205.385,A -85,B 0,C 180,E1 -2048.96,E2 -2048.96} C_VEL
LIN {X 0,Y 573.406,Z 216.467,A -85,B 0,C 180,E1 -2049.648,E2 -2049.648} C_VEL
LIN {X 0,Y 573.326,Z 227.261,A -85,B 0,C 180,E1 -2050.486,E2 -2050.486} C_VEL
LIN {X 0,Y 573.246,Z 236.828,A -85,B 0,C 180,E1 -2051.412,E2 -2051.412} C_VEL
LIN {X 0,Y 573.136,Z 246.043,A -85,B 0,C 180,E1 -2052.517,E2 -2052.517} C_VEL
LIN {X 0,Y 573.021,Z 253.339,A -85,B 0,C 180,E1 -2053.615,E2 -2053.615} C_VEL
LIN {X 0,Y 573.023,Z 259.107,A -85,B 0,C 180,E1 -2054.711,E2 -2054.711} C_VEL
LIN {X 0,Y 572.994,Z 263.59,A -85,B 0,C 180,E1 -2055.8,E2 -2055.8} C_VEL
LIN {X 0,Y 573.004,Z 265.945,A -85,B 0,C 180,E1 -2056.524,E2 -2056.524} C_VEL
LIN {X 0,Y 572.955,Z 267.837,A -85,B 0,C 180,E1 -2057.244,E2 -2057.244} C_VEL
LIN {X 0,Y 572.948,Z 269.242,A -85,B 0,C 180,E1 -2057.964,E2 -2057.964} C_VEL
LIN {X 0,Y 572.984,Z 270.462,A -85,B 0,C 180,E1 -2058.887,E2 -2058.887} C_VEL
LIN {X 0,Y 572.974,Z 270.991,A -85,B 0,C 180,E1 -2060.112,E2 -2060.112} C_VEL
LIN {X 0,Y 572.949,Z 270.087,A -85,B 0,C 180,E1 -2061.536,E2 -2061.536} C_VEL
LIN {X 0,Y 572.976,Z 269.049,A -85,B 0,C 180,E1 -2062.246,E2 -2062.246} C_VEL
LIN {X 0,Y 573.028,Z 266.342,A -85,B 0,C 180,E1 -2063.433,E2 -2063.433} C_VEL
LIN {X 0,Y 572.996,Z 261.952,A -85,B 0,C 180,E1 -2064.722,E2 -2064.722} C_VEL
LIN {X 0,Y 573.035,Z 257.145,A -85,B 0,C 180,E1 -2065.78,E2 -2065.78} C_VEL
LIN {X 0,Y 573.06,Z 251.102,A -85,B 0,C 180,E1 -2066.836,E2 -2066.836} C_VEL
LIN {X 0,Y 573.114,Z 243.612,A -85,B 0,C 180,E1 -2067.892,E2 -2067.892} C_VEL
LIN {X 0,Y 573.238,Z 235.981,A -85,B 0,C 180,E1 -2068.771,E2 -2068.771} C_VEL
LIN {X 0,Y 573.329,Z 225.68,A -85,B 0,C 180,E1 -2069.737,E2 -2069.737} C_VEL
LIN {X 0,Y 573.405,Z 215.236,A -85,B 0,C 180,E1 -2070.527,E2 -2070.527} C_VEL
LIN {X 0,Y 573.537,Z 203.589,A -85,B 0,C 180,E1 -2071.229,E2 -2071.229} C_VEL
LIN {X 0,Y 573.706,Z 191.166,A -85,B 0,C 180,E1 -2071.799,E2 -2071.799} C_VEL
LIN {X 0,Y 573.762,Z 178.12,A -85,B 0,C 180,E1 -2072.238,E2 -2072.238} C_VEL
LIN {X 0,Y 573.863,Z 164.794,A -85,B 0,C 180,E1 -2072.523,E2 -2072.523} C_VEL
LIN {X 0,Y 574.023,Z 65.816,A -85,B 0,C 180,E1 -2073.773,E2 -2073.773} C_VEL
LIN {X 0,Y 573.235,Z 60.84,A -85,B 0,C 180,E1 -2073.867,E2 -2073.867} C_VEL
LIN {X 0,Y 573.366,Z 48.193,A -85,B 0,C 180,E1 -2076.334,E2 -2076.334} C_VEL
LIN {X 0,Y 573.269,Z 41.076,A -85,B 0,C 180,E1 -2077.75,E2 -2077.75} C_VEL
LIN {X 0,Y 573.268,Z 41.08,A -85,B 0,C 180,E1 -2080.597,E2 -2080.597} C_VEL
LIN {X 0,Y 573.266,Z 41.08,A -85,B 0,C 180,E1 -2082.749,E2 -2082.749} C_VEL
LIN {X 0,Y 573.237,Z 41.079,A -85,B 0,C 180,E1 -2084.92,E2 -2084.92} C_VEL
LIN {X 0,Y 573.246,Z 41.075,A -85,B 0,C 180,E1 -2087.849,E2 -2087.849} C_VEL
LIN {X 0,Y 573.245,Z 41.079,A -85,B 0,C 180,E1 -2090.077,E2 -2090.077} C_VEL
LIN {X 0,Y 573.238,Z 41.084,A -85,B 0,C 180,E1 -2092.338,E2 -2092.338} C_VEL
LIN {X 0,Y 573.255,Z 41.073,A -85,B 0,C 180,E1 -2095.41,E2 -2095.41} C_VEL
LIN {X 0,Y 573.255,Z 41.081,A -85,B 0,C 180,E1 -2098.029,E2 -2098.029} C_VEL
LIN {X 0,Y 573.231,Z 41.076,A -85,B 0,C 180,E1 -2100.882,E2 -2100.882} C_VEL
LIN {X 0,Y 573.265,Z 41.075,A -85,B 0,C 180,E1 -2103.524,E2 -2103.524} C_VEL
LIN {X 0,Y 573.24,Z 41.08,A -85,B 0,C 180,E1 -2106.05,E2 -2106.05} C_VEL
LIN {X 0,Y 573.245,Z 41.074,A -85,B 0,C 180,E1 -2108.702,E2 -2108.702} C_VEL
LIN {X 0,Y 573.233,Z 41.085,A -85,B 0,C 180,E1 -2111.593,E2 -2111.593} C_VEL
LIN {X 0,Y 573.225,Z 41.076,A -85,B 0,C 180,E1 -2114.335,E2 -2114.335} C_VEL
LIN {X 0,Y 573.243,Z 41.083,A -85,B 0,C 180,E1 -2117.359,E2 -2117.359} C_VEL
LIN {X 0,Y 573.244,Z 41.074,A -85,B 0,C 180,E1 -2120.393,E2 -2120.393} C_VEL
LIN {X 0,Y 573.256,Z 41.08,A -85,B 0,C 180,E1 -2123.078,E2 -2123.078} C_VEL
LIN {X 0,Y 573.272,Z 41.072,A -85,B 0,C 180,E1 -2125.672,E2 -2125.672} C_VEL
LIN {X 0,Y 573.242,Z 41.074,A -85,B 0,C 180,E1 -2128.185,E2 -2128.185} C_VEL
LIN {X 0,Y 573.268,Z 41.076,A -85,B 0,C 180,E1 -2130.634,E2 -2130.634} C_VEL
LIN {X 0,Y 573.255,Z 41.079,A -85,B 0,C 180,E1 -2133.024,E2 -2133.024} C_VEL
LIN {X 0,Y 573.28,Z 41.071,A -85,B 0,C 180,E1 -2135.366,E2 -2135.366} C_VEL
LIN {X 0,Y 573.234,Z 41.081,A -85,B 0,C 180,E1 -2138.42,E2 -2138.42} C_VEL
LIN {X 0,Y 573.275,Z 41.077,A -85,B 0,C 180,E1 -2140.731,E2 -2140.731} C_VEL
LIN {X 0,Y 573.248,Z 41.074,A -85,B 0,C 180,E1 -2143.622,E2 -2143.622} C_VEL
LIN {X 0,Y 573.278,Z 41.072,A -85,B 0,C 180,E1 -2145.807,E2 -2145.807} C_VEL
LIN {X 0,Y 573.269,Z 41.073,A -85,B 0,C 180,E1 -2148.745,E2 -2148.745} C_VEL
LIN {X 0,Y 573.261,Z 41.073,A -85,B 0,C 180,E1 -2151.54,E2 -2151.54} C_VEL
LIN {X 0,Y 573.25,Z 41.077,A -85,B 0,C 180,E1 -2153.665,E2 -2153.665} C_VEL
LIN {X 0,Y 573.229,Z 41.082,A -85,B 0,C 180,E1 -2155.781,E2 -2155.781} C_VEL
LIN {X 0,Y 573.312,Z 41.075,A -85,B 0,C 180,E1 -2157.893,E2 -2157.893} C_VEL
LIN {X 0,Y 573.333,Z 41.063,A -85,B 0,C 180,E1 -2160.702,E2 -2160.702} C_VEL
LIN {X 0,Y 573.235,Z 41.081,A -85,B 0,C 180,E1 -2163.515,E2 -2163.515} C_VEL
LIN {X 0,Y 573.287,Z 41.078,A -85,B 0,C 180,E1 -2165.628,E2 -2165.628} C_VEL
LIN {X 0,Y 573.259,Z 41.072,A -85,B 0,C 180,E1 -2168.46,E2 -2168.46} C_VEL
LIN {X 0,Y 573.279,Z 41.077,A -85,B 0,C 180,E1 -2171.312,E2 -2171.312} C_VEL
LIN {X 0,Y 573.282,Z 41.069,A -85,B 0,C 180,E1 -2174.422,E2 -2174.422} C_VEL
LIN {X 0,Y 573.264,Z 41.079,A -85,B 0,C 180,E1 -2177.112,E2 -2177.112} C_VEL
LIN {X 0,Y 573.246,Z 41.074,A -85,B 0,C 180,E1 -2180.077,E2 -2180.077} C_VEL
LIN {X 0,Y 573.238,Z 41.075,A -85,B 0,C 180,E1 -2182.338,E2 -2182.338} C_VEL
LIN {X 0,Y 573.25,Z 41.076,A -85,B 0,C 180,E1 -2185.41,E2 -2185.41} C_VEL
LIN {X 0,Y 573.234,Z 41.081,A -85,B 0,C 180,E1 -2188.565,E2 -2188.565} C_VEL
LIN {X 0,Y 573.229,Z 41.081,A -85,B 0,C 180,E1 -2190.993,E2 -2190.993} C_VEL
LIN {X 0,Y 573.246,Z 41.074,A -85,B 0,C 180,E1 -2193.521,E2 -2193.521} C_VEL
LIN {X 0,Y 573.198,Z 41.082,A -85,B 0,C 180,E1 -2196.053,E2 -2196.053} C_VEL
LIN {X 0,Y 573.242,Z 41.08,A -85,B 0,C 180,E1 -2198.702,E2 -2198.702} C_VEL
LIN {X 0,Y 573.233,Z 41.076,A -85,B 0,C 180,E1 -2201.593,E2 -2201.593} C_VEL
LIN {X 0,Y 573.227,Z 41.085,A -85,B 0,C 180,E1 -2204.335,E2 -2204.335} C_VEL
LIN {X 0,Y 573.24,Z 41.075,A -85,B 0,C 180,E1 -2207.359,E2 -2207.359} C_VEL
LIN {X 0,Y 573.24,Z 41.079,A -85,B 0,C 180,E1 -2210.392,E2 -2210.392} C_VEL
LIN {X 0,Y 573.236,Z 41.075,A -85,B 0,C 180,E1 -2213.076,E2 -2213.076} C_VEL
LIN {X 0,Y 573.266,Z 41.078,A -85,B 0,C 180,E1 -2215.671,E2 -2215.671} C_VEL
LIN {X 0,Y 573.242,Z 41.077,A -85,B 0,C 180,E1 -2218.184,E2 -2218.184} C_VEL
LIN {X 0,Y 573.262,Z 41.073,A -85,B 0,C 180,E1 -2220.634,E2 -2220.634} C_VEL
LIN {X 0,Y 573.239,Z 41.084,A -85,B 0,C 180,E1 -2223.508,E2 -2223.508} C_VEL
LIN {X 0,Y 573.296,Z 41.243,A -85,B 0,C 180,E1 -2225.825,E2 -2225.825} C_VEL
LIN {X 0,Y 573.997,Z 45.789,A -85,B 0,C 180,E1 -2226.476,E2 -2226.476} C_VEL
LIN {X 0,Y 573.813,Z 65.874,A -85,B 0,C 180,E1 -2229.195,E2 -2229.195} C_VEL
LIN {X 0,Y 573.699,Z 85.394,A -85,B 0,C 180,E1 -2231.797,E2 -2231.797} C_VEL
LIN {X 0,Y 573.52,Z 106.156,A -85,B 0,C 180,E1 -2234.542,E2 -2234.542} C_VEL
LIN {X 0,Y 573.439,Z 118.353,A -85,B 0,C 180,E1 -2236.162,E2 -2236.162} C_VEL
LIN {X 0,Y 574.062,Z 124.494,A -85,B 0,C 180,E1 -2236.256,E2 -2236.256} C_VEL
LIN {X 0,Y 573.85,Z 226.938,A -85,B 0,C 180,E1 -2237.557,E2 -2237.557} C_VEL
LIN {X 0,Y 573.802,Z 240.212,A -85,B 0,C 180,E1 -2237.87,E2 -2237.87} C_VEL
LIN {X 0,Y 573.71,Z 252.374,A -85,B 0,C 180,E1 -2238.294,E2 -2238.294} C_VEL
LIN {X 0,Y 573.586,Z 264.66,A -85,B 0,C 180,E1 -2238.875,E2 -2238.875} C_VEL
LIN {X 0,Y 573.425,Z 276.195,A -85,B 0,C 180,E1 -2239.585,E2 -2239.585} C_VEL
LIN {X 0,Y 573.333,Z 286.602,A -85,B 0,C 180,E1 -2240.385,E2 -2240.385} C_VEL
LIN {X 0,Y 573.241,Z 295.112,A -85,B 0,C 180,E1 -2241.184,E2 -2241.184} C_VEL
LIN {X 0,Y 573.161,Z 302.96,A -85,B 0,C 180,E1 -2242.071,E2 -2242.071} C_VEL
LIN {X 0,Y 573.073,Z 310.955,A -85,B 0,C 180,E1 -2243.185,E2 -2243.185} C_VEL
LIN {X 0,Y 573.07,Z 317.679,A -85,B 0,C 180,E1 -2244.37,E2 -2244.37} C_VEL
LIN {X 0,Y 573.028,Z 322.372,A -85,B 0,C 180,E1 -2245.427,E2 -2245.427} C_VEL
LIN {X 0,Y 573.022,Z 325.958,A -85,B 0,C 180,E1 -2246.484,E2 -2246.484} C_VEL
LIN {X 0,Y 572.959,Z 327.807,A -85,B 0,C 180,E1 -2247.188,E2 -2247.188} C_VEL
LIN {X 0,Y 572.946,Z 330.184,A -85,B 0,C 180,E1 -2248.594,E2 -2248.594} C_VEL
LIN {X 0,Y 572.938,Z 331,A -85,B 0,C 180,E1 -2250,E2 -2250} C_VEL
LIN {X 0,Y 572.946,Z 330.185,A -85,B 0,C 180,E1 -2251.406,E2 -2251.406} C_VEL
LIN {X 0,Y 572.959,Z 327.81,A -85,B 0,C 180,E1 -2252.812,E2 -2252.812} C_VEL
LIN {X 0,Y 573.015,Z 324.896,A -85,B 0,C 180,E1 -2253.868,E2 -2253.868} C_VEL
LIN {X 0,Y 572.963,Z 320.949,A -85,B 0,C 180,E1 -2254.926,E2 -2254.926} C_VEL
LIN {X 0,Y 573.093,Z 315.867,A -85,B 0,C 180,E1 -2255.983,E2 -2255.983} C_VEL
LIN {X 0,Y 573.103,Z 309.468,A -85,B 0,C 180,E1 -2257.044,E2 -2257.044} C_VEL
LIN {X 0,Y 573.177,Z 301.478,A -85,B 0,C 180,E1 -2258.106,E2 -2258.106} C_VEL
LIN {X 0,Y 573.254,Z 293.334,A -85,B 0,C 180,E1 -2258.993,E2 -2258.993} C_VEL
LIN {X 0,Y 573.344,Z 283.399,A -85,B 0,C 180,E1 -2259.881,E2 -2259.881} C_VEL
LIN {X 0,Y 573.501,Z 272.21,A -85,B 0,C 180,E1 -2260.679,E2 -2260.679} C_VEL
LIN {X 0,Y 573.586,Z 261.173,A -85,B 0,C 180,E1 -2261.306,E2 -2261.306} C_VEL
LIN {X 0,Y 573.709,Z 248.978,A -85,B 0,C 180,E1 -2261.84,E2 -2261.84} C_VEL
LIN {X 0,Y 573.812,Z 236.172,A -85,B 0,C 180,E1 -2262.242,E2 -2262.242} C_VEL
LIN {X 0,Y 573.909,Z 222.597,A -85,B 0,C 180,E1 -2262.509,E2 -2262.509} C_VEL
LIN {X 0,Y 573.94,Z 121.945,A -85,B 0,C 180,E1 -2263.779,E2 -2263.779} C_VEL
LIN {X 0,Y 573.441,Z 118.269,A -85,B 0,C 180,E1 -2263.85,E2 -2263.85} C_VEL
LIN {X 0,Y 573.6,Z 96.528,A -85,B 0,C 180,E1 -2266.731,E2 -2266.731} C_VEL
LIN {X 0,Y 573.722,Z 76.365,A -85,B 0,C 180,E1 -2269.397,E2 -2269.397} C_VEL
LIN {X 0,Y 573.894,Z 54.638,A -85,B 0,C 180,E1 -2272.311,E2 -2272.311} C_VEL
LIN {X 0,Y 573.904,Z 44.593,A -85,B 0,C 180,E1 -2273.682,E2 -2273.682} C_VEL
LIN {X 0,Y 573.273,Z 41.079,A -85,B 0,C 180,E1 -2274.2,E2 -2274.2} C_VEL
LIN {X 0,Y 573.252,Z 41.076,A -85,B 0,C 180,E1 -2276.976,E2 -2276.976} C_VEL
LIN {X 0,Y 573.249,Z 41.074,A -85,B 0,C 180,E1 -2279.488,E2 -2279.488} C_VEL
LIN {X 0,Y 573.256,Z 41.076,A -85,B 0,C 180,E1 -2282.645,E2 -2282.645} C_VEL
LIN {X 0,Y 573.211,Z 41.079,A -85,B 0,C 180,E1 -2285.188,E2 -2285.188} C_VEL
LIN {X 0,Y 573.238,Z 41.082,A -85,B 0,C 180,E1 -2287.808,E2 -2287.808} C_VEL
LIN {X 0,Y 573.248,Z 41.075,A -85,B 0,C 180,E1 -2290.525,E2 -2290.525} C_VEL
LIN {X 0,Y 573.239,Z 41.078,A -85,B 0,C 180,E1 -2293.359,E2 -2293.359} C_VEL
LIN {X 0,Y 573.24,Z 41.074,A -85,B 0,C 180,E1 -2296.641,E2 -2296.641} C_VEL
